BEGIN
   BB_G1.Bef.Bed_Res := FALSE;
   BB_G1.Bef.Bed_UV := FALSE;
   BB_G1.Bef.Bed_NHV := FALSE;
   BB_G1.Bef.Bed_PLS := FALSE;
   BB_G1.Bef.BA_Hand := FALSE;
   BB_G1.Bef.BA_Auto := FALSE;
   BB_G1.Bef.BF_Ein1 := FALSE;
   BB_G1.Bef.BF_Ein2 := FALSE;
   BB_G1.Bef.BF_Aus := FALSE;
   BB_G1.Bef.BZ_Res := FALSE;
   BB_G1.Bef.Res_10 := FALSE;
   BB_G1.Bef.Res_11 := FALSE;
   BB_G1.Bef.Res_12 := FALSE;
   BB_G1.Bef.Res_13 := FALSE;
   BB_G1.Bef.Res_14 := FALSE;
   BB_G1.Bef.Res_15 := FALSE;
   BB_G1.Bef.Res_16 := FALSE;
   BB_G1.Bef.Res_17 := FALSE;
   BB_G1.Bef.Res_18 := FALSE;
   BB_G1.Bef.Res_19 := FALSE;
   BB_G1.Bef.Res_20 := FALSE;
   BB_G1.Bef.Res_21 := FALSE;
   BB_G1.Bef.Res_22 := FALSE;
   BB_G1.Bef.Res_23 := FALSE;
   BB_G1.Bef.Res_24 := FALSE;
   BB_G1.Bef.Res_25 := FALSE;
   BB_G1.Bef.Res_26 := FALSE;
   BB_G1.Bef.Res_27 := FALSE;
   BB_G1.Bef.Res_28 := FALSE;
   BB_G1.Bef.Res_29 := FALSE;
   BB_G1.Bef.BF_Set_SW_chg := FALSE;
   BB_G1.Bef.BF_Quit := FALSE;
   BB_G1.SW_Hand := 0.0;
   BB_G2.Bef.Bed_Res := FALSE;
   BB_G2.Bef.Bed_UV := FALSE;
   BB_G2.Bef.Bed_NHV := FALSE;
   BB_G2.Bef.Bed_PLS := FALSE;
   BB_G2.Bef.BA_Hand := FALSE;
   BB_G2.Bef.BA_Auto := FALSE;
   BB_G2.Bef.BF_Ein1 := FALSE;
   BB_G2.Bef.BF_Ein2 := FALSE;
   BB_G2.Bef.BF_Aus := FALSE;
   BB_G2.Bef.BZ_Res := FALSE;
   BB_G2.Bef.Res_10 := FALSE;
   BB_G2.Bef.Res_11 := FALSE;
   BB_G2.Bef.Res_12 := FALSE;
   BB_G2.Bef.Res_13 := FALSE;
   BB_G2.Bef.Res_14 := FALSE;
   BB_G2.Bef.Res_15 := FALSE;
   BB_G2.Bef.Res_16 := FALSE;
   BB_G2.Bef.Res_17 := FALSE;
   BB_G2.Bef.Res_18 := FALSE;
   BB_G2.Bef.Res_19 := FALSE;
   BB_G2.Bef.Res_20 := FALSE;
   BB_G2.Bef.Res_21 := FALSE;
   BB_G2.Bef.Res_22 := FALSE;
   BB_G2.Bef.Res_23 := FALSE;
   BB_G2.Bef.Res_24 := FALSE;
   BB_G2.Bef.Res_25 := FALSE;
   BB_G2.Bef.Res_26 := FALSE;
   BB_G2.Bef.Res_27 := FALSE;
   BB_G2.Bef.Res_28 := FALSE;
   BB_G2.Bef.Res_29 := FALSE;
   BB_G2.Bef.BF_Set_SW_chg := FALSE;
   BB_G2.Bef.BF_Quit := FALSE;
   BB_G2.SW_Hand := 0.0;
   BB_G3.Bef.Bed_Res := FALSE;
   BB_G3.Bef.Bed_UV := FALSE;
   BB_G3.Bef.Bed_NHV := FALSE;
   BB_G3.Bef.Bed_PLS := FALSE;
   BB_G3.Bef.BA_Hand := FALSE;
   BB_G3.Bef.BA_Auto := FALSE;
   BB_G3.Bef.BF_Ein1 := FALSE;
   BB_G3.Bef.BF_Ein2 := FALSE;
   BB_G3.Bef.BF_Aus := FALSE;
   BB_G3.Bef.BZ_Res := FALSE;
   BB_G3.Bef.Res_10 := FALSE;
   BB_G3.Bef.Res_11 := FALSE;
   BB_G3.Bef.Res_12 := FALSE;
   BB_G3.Bef.Res_13 := FALSE;
   BB_G3.Bef.Res_14 := FALSE;
   BB_G3.Bef.Res_15 := FALSE;
   BB_G3.Bef.Res_16 := FALSE;
   BB_G3.Bef.Res_17 := FALSE;
   BB_G3.Bef.Res_18 := FALSE;
   BB_G3.Bef.Res_19 := FALSE;
   BB_G3.Bef.Res_20 := FALSE;
   BB_G3.Bef.Res_21 := FALSE;
   BB_G3.Bef.Res_22 := FALSE;
   BB_G3.Bef.Res_23 := FALSE;
   BB_G3.Bef.Res_24 := FALSE;
   BB_G3.Bef.Res_25 := FALSE;
   BB_G3.Bef.Res_26 := FALSE;
   BB_G3.Bef.Res_27 := FALSE;
   BB_G3.Bef.Res_28 := FALSE;
   BB_G3.Bef.Res_29 := FALSE;
   BB_G3.Bef.BF_Set_SW_chg := FALSE;
   BB_G3.Bef.BF_Quit := FALSE;
   BB_G3.SW_Hand := 0.0;
   BB_SHL_G1.Bef.Bed_Res := FALSE;
   BB_SHL_G1.Bef.Bed_UV := FALSE;
   BB_SHL_G1.Bef.Bed_NHV := FALSE;
   BB_SHL_G1.Bef.Bed_PLS := FALSE;
   BB_SHL_G1.Bef.BA_Hand := FALSE;
   BB_SHL_G1.Bef.BA_Auto := FALSE;
   BB_SHL_G1.Bef.BF_Ein1 := FALSE;
   BB_SHL_G1.Bef.BF_Ein2 := FALSE;
   BB_SHL_G1.Bef.BF_Aus := FALSE;
   BB_SHL_G1.Bef.BZ_Res := FALSE;
   BB_SHL_G1.Bef.Res_10 := FALSE;
   BB_SHL_G1.Bef.Res_11 := FALSE;
   BB_SHL_G1.Bef.Res_12 := FALSE;
   BB_SHL_G1.Bef.Res_13 := FALSE;
   BB_SHL_G1.Bef.Res_14 := FALSE;
   BB_SHL_G1.Bef.Res_15 := FALSE;
   BB_SHL_G1.Bef.Res_16 := FALSE;
   BB_SHL_G1.Bef.Res_17 := FALSE;
   BB_SHL_G1.Bef.Res_18 := FALSE;
   BB_SHL_G1.Bef.Res_19 := FALSE;
   BB_SHL_G1.Bef.Res_20 := FALSE;
   BB_SHL_G1.Bef.Res_21 := FALSE;
   BB_SHL_G1.Bef.Res_22 := FALSE;
   BB_SHL_G1.Bef.Res_23 := FALSE;
   BB_SHL_G1.Bef.Res_24 := FALSE;
   BB_SHL_G1.Bef.Res_25 := FALSE;
   BB_SHL_G1.Bef.Res_26 := FALSE;
   BB_SHL_G1.Bef.Res_27 := FALSE;
   BB_SHL_G1.Bef.Res_28 := FALSE;
   BB_SHL_G1.Bef.Res_29 := FALSE;
   BB_SHL_G1.Bef.BF_Set_SW_chg := FALSE;
   BB_SHL_G1.Bef.BF_Quit := FALSE;
   BB_SHL_G1.SW_Hand := 0.0;
   BB_SHL_G2.Bef.Bed_Res := FALSE;
   BB_SHL_G2.Bef.Bed_UV := FALSE;
   BB_SHL_G2.Bef.Bed_NHV := FALSE;
   BB_SHL_G2.Bef.Bed_PLS := FALSE;
   BB_SHL_G2.Bef.BA_Hand := FALSE;
   BB_SHL_G2.Bef.BA_Auto := FALSE;
   BB_SHL_G2.Bef.BF_Ein1 := FALSE;
   BB_SHL_G2.Bef.BF_Ein2 := FALSE;
   BB_SHL_G2.Bef.BF_Aus := FALSE;
   BB_SHL_G2.Bef.BZ_Res := FALSE;
   BB_SHL_G2.Bef.Res_10 := FALSE;
   BB_SHL_G2.Bef.Res_11 := FALSE;
   BB_SHL_G2.Bef.Res_12 := FALSE;
   BB_SHL_G2.Bef.Res_13 := FALSE;
   BB_SHL_G2.Bef.Res_14 := FALSE;
   BB_SHL_G2.Bef.Res_15 := FALSE;
   BB_SHL_G2.Bef.Res_16 := FALSE;
   BB_SHL_G2.Bef.Res_17 := FALSE;
   BB_SHL_G2.Bef.Res_18 := FALSE;
   BB_SHL_G2.Bef.Res_19 := FALSE;
   BB_SHL_G2.Bef.Res_20 := FALSE;
   BB_SHL_G2.Bef.Res_21 := FALSE;
   BB_SHL_G2.Bef.Res_22 := FALSE;
   BB_SHL_G2.Bef.Res_23 := FALSE;
   BB_SHL_G2.Bef.Res_24 := FALSE;
   BB_SHL_G2.Bef.Res_25 := FALSE;
   BB_SHL_G2.Bef.Res_26 := FALSE;
   BB_SHL_G2.Bef.Res_27 := FALSE;
   BB_SHL_G2.Bef.Res_28 := FALSE;
   BB_SHL_G2.Bef.Res_29 := FALSE;
   BB_SHL_G2.Bef.BF_Set_SW_chg := FALSE;
   BB_SHL_G2.Bef.BF_Quit := FALSE;
   BB_SHL_G2.SW_Hand := 0.0;
   BB_SHL_G3.Bef.Bed_Res := FALSE;
   BB_SHL_G3.Bef.Bed_UV := FALSE;
   BB_SHL_G3.Bef.Bed_NHV := FALSE;
   BB_SHL_G3.Bef.Bed_PLS := FALSE;
   BB_SHL_G3.Bef.BA_Hand := FALSE;
   BB_SHL_G3.Bef.BA_Auto := FALSE;
   BB_SHL_G3.Bef.BF_Ein1 := FALSE;
   BB_SHL_G3.Bef.BF_Ein2 := FALSE;
   BB_SHL_G3.Bef.BF_Aus := FALSE;
   BB_SHL_G3.Bef.BZ_Res := FALSE;
   BB_SHL_G3.Bef.Res_10 := FALSE;
   BB_SHL_G3.Bef.Res_11 := FALSE;
   BB_SHL_G3.Bef.Res_12 := FALSE;
   BB_SHL_G3.Bef.Res_13 := FALSE;
   BB_SHL_G3.Bef.Res_14 := FALSE;
   BB_SHL_G3.Bef.Res_15 := FALSE;
   BB_SHL_G3.Bef.Res_16 := FALSE;
   BB_SHL_G3.Bef.Res_17 := FALSE;
   BB_SHL_G3.Bef.Res_18 := FALSE;
   BB_SHL_G3.Bef.Res_19 := FALSE;
   BB_SHL_G3.Bef.Res_20 := FALSE;
   BB_SHL_G3.Bef.Res_21 := FALSE;
   BB_SHL_G3.Bef.Res_22 := FALSE;
   BB_SHL_G3.Bef.Res_23 := FALSE;
   BB_SHL_G3.Bef.Res_24 := FALSE;
   BB_SHL_G3.Bef.Res_25 := FALSE;
   BB_SHL_G3.Bef.Res_26 := FALSE;
   BB_SHL_G3.Bef.Res_27 := FALSE;
   BB_SHL_G3.Bef.Res_28 := FALSE;
   BB_SHL_G3.Bef.Res_29 := FALSE;
   BB_SHL_G3.Bef.BF_Set_SW_chg := FALSE;
   BB_SHL_G3.Bef.BF_Quit := FALSE;
   BB_SHL_G3.SW_Hand := 0.0;
   BB_AV.Bef.Bed_Res := FALSE;
   BB_AV.Bef.Bed_UV := FALSE;
   BB_AV.Bef.Bed_NHV := FALSE;
   BB_AV.Bef.Bed_PLS := FALSE;
   BB_AV.Bef.BA_Hand := FALSE;
   BB_AV.Bef.BA_Auto := FALSE;
   BB_AV.Bef.BF_Ein1 := FALSE;
   BB_AV.Bef.BF_Ein2 := FALSE;
   BB_AV.Bef.BF_Aus := FALSE;
   BB_AV.Bef.BZ_Res := FALSE;
   BB_AV.Bef.Res_10 := FALSE;
   BB_AV.Bef.Res_11 := FALSE;
   BB_AV.Bef.Res_12 := FALSE;
   BB_AV.Bef.Res_13 := FALSE;
   BB_AV.Bef.Res_14 := FALSE;
   BB_AV.Bef.Res_15 := FALSE;
   BB_AV.Bef.Res_16 := FALSE;
   BB_AV.Bef.Res_17 := FALSE;
   BB_AV.Bef.Res_18 := FALSE;
   BB_AV.Bef.Res_19 := FALSE;
   BB_AV.Bef.Res_20 := FALSE;
   BB_AV.Bef.Res_21 := FALSE;
   BB_AV.Bef.Res_22 := FALSE;
   BB_AV.Bef.Res_23 := FALSE;
   BB_AV.Bef.Res_24 := FALSE;
   BB_AV.Bef.Res_25 := FALSE;
   BB_AV.Bef.Res_26 := FALSE;
   BB_AV.Bef.Res_27 := FALSE;
   BB_AV.Bef.Res_28 := FALSE;
   BB_AV.Bef.Res_29 := FALSE;
   BB_AV.Bef.BF_Set_SW_chg := FALSE;
   BB_AV.Bef.BF_Quit := FALSE;
   BB_AV.SW_Hand := 0.0;
   BB_LS1.Bef.Bed_Res := FALSE;
   BB_LS1.Bef.Bed_UV := FALSE;
   BB_LS1.Bef.Bed_NHV := FALSE;
   BB_LS1.Bef.Bed_PLS := FALSE;
   BB_LS1.Bef.BA_Hand := FALSE;
   BB_LS1.Bef.BA_Auto := FALSE;
   BB_LS1.Bef.BF_Ein1 := FALSE;
   BB_LS1.Bef.BF_Ein2 := FALSE;
   BB_LS1.Bef.BF_Aus := FALSE;
   BB_LS1.Bef.BZ_Res := FALSE;
   BB_LS1.Bef.Res_10 := FALSE;
   BB_LS1.Bef.Res_11 := FALSE;
   BB_LS1.Bef.Res_12 := FALSE;
   BB_LS1.Bef.Res_13 := FALSE;
   BB_LS1.Bef.Res_14 := FALSE;
   BB_LS1.Bef.Res_15 := FALSE;
   BB_LS1.Bef.Res_16 := FALSE;
   BB_LS1.Bef.Res_17 := FALSE;
   BB_LS1.Bef.Res_18 := FALSE;
   BB_LS1.Bef.Res_19 := FALSE;
   BB_LS1.Bef.Res_20 := FALSE;
   BB_LS1.Bef.Res_21 := FALSE;
   BB_LS1.Bef.Res_22 := FALSE;
   BB_LS1.Bef.Res_23 := FALSE;
   BB_LS1.Bef.Res_24 := FALSE;
   BB_LS1.Bef.Res_25 := FALSE;
   BB_LS1.Bef.Res_26 := FALSE;
   BB_LS1.Bef.Res_27 := FALSE;
   BB_LS1.Bef.Res_28 := FALSE;
   BB_LS1.Bef.Res_29 := FALSE;
   BB_LS1.Bef.BF_Set_SW_chg := FALSE;
   BB_LS1.Bef.BF_Quit := FALSE;
   BB_LS1.SW_Hand := 0.0;
   BB_LS2.Bef.Bed_Res := FALSE;
   BB_LS2.Bef.Bed_UV := FALSE;
   BB_LS2.Bef.Bed_NHV := FALSE;
   BB_LS2.Bef.Bed_PLS := FALSE;
   BB_LS2.Bef.BA_Hand := FALSE;
   BB_LS2.Bef.BA_Auto := FALSE;
   BB_LS2.Bef.BF_Ein1 := FALSE;
   BB_LS2.Bef.BF_Ein2 := FALSE;
   BB_LS2.Bef.BF_Aus := FALSE;
   BB_LS2.Bef.BZ_Res := FALSE;
   BB_LS2.Bef.Res_10 := FALSE;
   BB_LS2.Bef.Res_11 := FALSE;
   BB_LS2.Bef.Res_12 := FALSE;
   BB_LS2.Bef.Res_13 := FALSE;
   BB_LS2.Bef.Res_14 := FALSE;
   BB_LS2.Bef.Res_15 := FALSE;
   BB_LS2.Bef.Res_16 := FALSE;
   BB_LS2.Bef.Res_17 := FALSE;
   BB_LS2.Bef.Res_18 := FALSE;
   BB_LS2.Bef.Res_19 := FALSE;
   BB_LS2.Bef.Res_20 := FALSE;
   BB_LS2.Bef.Res_21 := FALSE;
   BB_LS2.Bef.Res_22 := FALSE;
   BB_LS2.Bef.Res_23 := FALSE;
   BB_LS2.Bef.Res_24 := FALSE;
   BB_LS2.Bef.Res_25 := FALSE;
   BB_LS2.Bef.Res_26 := FALSE;
   BB_LS2.Bef.Res_27 := FALSE;
   BB_LS2.Bef.Res_28 := FALSE;
   BB_LS2.Bef.Res_29 := FALSE;
   BB_LS2.Bef.BF_Set_SW_chg := FALSE;
   BB_LS2.Bef.BF_Quit := FALSE;
   BB_LS2.SW_Hand := 0.0;
   BB1_RZP1.Bef.Bed_Res := FALSE;
   BB1_RZP1.Bef.Bed_UV := FALSE;
   BB1_RZP1.Bef.Bed_NHV := FALSE;
   BB1_RZP1.Bef.Bed_PLS := FALSE;
   BB1_RZP1.Bef.BA_Hand := FALSE;
   BB1_RZP1.Bef.BA_Auto := FALSE;
   BB1_RZP1.Bef.BF_Ein1 := FALSE;
   BB1_RZP1.Bef.BF_Ein2 := FALSE;
   BB1_RZP1.Bef.BF_Aus := FALSE;
   BB1_RZP1.Bef.BZ_Res := FALSE;
   BB1_RZP1.Bef.Res_10 := FALSE;
   BB1_RZP1.Bef.Res_11 := FALSE;
   BB1_RZP1.Bef.Res_12 := FALSE;
   BB1_RZP1.Bef.Res_13 := FALSE;
   BB1_RZP1.Bef.Res_14 := FALSE;
   BB1_RZP1.Bef.Res_15 := FALSE;
   BB1_RZP1.Bef.Res_16 := FALSE;
   BB1_RZP1.Bef.Res_17 := FALSE;
   BB1_RZP1.Bef.Res_18 := FALSE;
   BB1_RZP1.Bef.Res_19 := FALSE;
   BB1_RZP1.Bef.Res_20 := FALSE;
   BB1_RZP1.Bef.Res_21 := FALSE;
   BB1_RZP1.Bef.Res_22 := FALSE;
   BB1_RZP1.Bef.Res_23 := FALSE;
   BB1_RZP1.Bef.Res_24 := FALSE;
   BB1_RZP1.Bef.Res_25 := FALSE;
   BB1_RZP1.Bef.Res_26 := FALSE;
   BB1_RZP1.Bef.Res_27 := FALSE;
   BB1_RZP1.Bef.Res_28 := FALSE;
   BB1_RZP1.Bef.Res_29 := FALSE;
   BB1_RZP1.Bef.BF_Set_SW_chg := FALSE;
   BB1_RZP1.Bef.BF_Quit := FALSE;
   BB1_RZP1.SW_Hand := 0.0;
   BB1_RZP2.Bef.Bed_Res := FALSE;
   BB1_RZP2.Bef.Bed_UV := FALSE;
   BB1_RZP2.Bef.Bed_NHV := FALSE;
   BB1_RZP2.Bef.Bed_PLS := FALSE;
   BB1_RZP2.Bef.BA_Hand := FALSE;
   BB1_RZP2.Bef.BA_Auto := FALSE;
   BB1_RZP2.Bef.BF_Ein1 := FALSE;
   BB1_RZP2.Bef.BF_Ein2 := FALSE;
   BB1_RZP2.Bef.BF_Aus := FALSE;
   BB1_RZP2.Bef.BZ_Res := FALSE;
   BB1_RZP2.Bef.Res_10 := FALSE;
   BB1_RZP2.Bef.Res_11 := FALSE;
   BB1_RZP2.Bef.Res_12 := FALSE;
   BB1_RZP2.Bef.Res_13 := FALSE;
   BB1_RZP2.Bef.Res_14 := FALSE;
   BB1_RZP2.Bef.Res_15 := FALSE;
   BB1_RZP2.Bef.Res_16 := FALSE;
   BB1_RZP2.Bef.Res_17 := FALSE;
   BB1_RZP2.Bef.Res_18 := FALSE;
   BB1_RZP2.Bef.Res_19 := FALSE;
   BB1_RZP2.Bef.Res_20 := FALSE;
   BB1_RZP2.Bef.Res_21 := FALSE;
   BB1_RZP2.Bef.Res_22 := FALSE;
   BB1_RZP2.Bef.Res_23 := FALSE;
   BB1_RZP2.Bef.Res_24 := FALSE;
   BB1_RZP2.Bef.Res_25 := FALSE;
   BB1_RZP2.Bef.Res_26 := FALSE;
   BB1_RZP2.Bef.Res_27 := FALSE;
   BB1_RZP2.Bef.Res_28 := FALSE;
   BB1_RZP2.Bef.Res_29 := FALSE;
   BB1_RZP2.Bef.BF_Set_SW_chg := FALSE;
   BB1_RZP2.Bef.BF_Quit := FALSE;
   BB1_RZP2.SW_Hand := 0.0;
   BB1_UeSP.Bef.Bed_Res := FALSE;
   BB1_UeSP.Bef.Bed_UV := FALSE;
   BB1_UeSP.Bef.Bed_NHV := FALSE;
   BB1_UeSP.Bef.Bed_PLS := FALSE;
   BB1_UeSP.Bef.BA_Hand := FALSE;
   BB1_UeSP.Bef.BA_Auto := FALSE;
   BB1_UeSP.Bef.BF_Ein1 := FALSE;
   BB1_UeSP.Bef.BF_Ein2 := FALSE;
   BB1_UeSP.Bef.BF_Aus := FALSE;
   BB1_UeSP.Bef.BZ_Res := FALSE;
   BB1_UeSP.Bef.Res_10 := FALSE;
   BB1_UeSP.Bef.Res_11 := FALSE;
   BB1_UeSP.Bef.Res_12 := FALSE;
   BB1_UeSP.Bef.Res_13 := FALSE;
   BB1_UeSP.Bef.Res_14 := FALSE;
   BB1_UeSP.Bef.Res_15 := FALSE;
   BB1_UeSP.Bef.Res_16 := FALSE;
   BB1_UeSP.Bef.Res_17 := FALSE;
   BB1_UeSP.Bef.Res_18 := FALSE;
   BB1_UeSP.Bef.Res_19 := FALSE;
   BB1_UeSP.Bef.Res_20 := FALSE;
   BB1_UeSP.Bef.Res_21 := FALSE;
   BB1_UeSP.Bef.Res_22 := FALSE;
   BB1_UeSP.Bef.Res_23 := FALSE;
   BB1_UeSP.Bef.Res_24 := FALSE;
   BB1_UeSP.Bef.Res_25 := FALSE;
   BB1_UeSP.Bef.Res_26 := FALSE;
   BB1_UeSP.Bef.Res_27 := FALSE;
   BB1_UeSP.Bef.Res_28 := FALSE;
   BB1_UeSP.Bef.Res_29 := FALSE;
   BB1_UeSP.Bef.BF_Set_SW_chg := FALSE;
   BB1_UeSP.Bef.BF_Quit := FALSE;
   BB1_UeSP.SW_Hand := 0.0;
   BB1_AS1.Bef.Bed_Res := FALSE;
   BB1_AS1.Bef.Bed_UV := FALSE;
   BB1_AS1.Bef.Bed_NHV := FALSE;
   BB1_AS1.Bef.Bed_PLS := FALSE;
   BB1_AS1.Bef.BA_Hand := FALSE;
   BB1_AS1.Bef.BA_Auto := FALSE;
   BB1_AS1.Bef.BF_Ein1 := FALSE;
   BB1_AS1.Bef.BF_Ein2 := FALSE;
   BB1_AS1.Bef.BF_Aus := FALSE;
   BB1_AS1.Bef.BZ_Res := FALSE;
   BB1_AS1.Bef.Res_10 := FALSE;
   BB1_AS1.Bef.Res_11 := FALSE;
   BB1_AS1.Bef.Res_12 := FALSE;
   BB1_AS1.Bef.Res_13 := FALSE;
   BB1_AS1.Bef.Res_14 := FALSE;
   BB1_AS1.Bef.Res_15 := FALSE;
   BB1_AS1.Bef.Res_16 := FALSE;
   BB1_AS1.Bef.Res_17 := FALSE;
   BB1_AS1.Bef.Res_18 := FALSE;
   BB1_AS1.Bef.Res_19 := FALSE;
   BB1_AS1.Bef.Res_20 := FALSE;
   BB1_AS1.Bef.Res_21 := FALSE;
   BB1_AS1.Bef.Res_22 := FALSE;
   BB1_AS1.Bef.Res_23 := FALSE;
   BB1_AS1.Bef.Res_24 := FALSE;
   BB1_AS1.Bef.Res_25 := FALSE;
   BB1_AS1.Bef.Res_26 := FALSE;
   BB1_AS1.Bef.Res_27 := FALSE;
   BB1_AS1.Bef.Res_28 := FALSE;
   BB1_AS1.Bef.Res_29 := FALSE;
   BB1_AS1.Bef.BF_Set_SW_chg := FALSE;
   BB1_AS1.Bef.BF_Quit := FALSE;
   BB1_AS1.SW_Hand := 0.0;
   BB1_AS2.Bef.Bed_Res := FALSE;
   BB1_AS2.Bef.Bed_UV := FALSE;
   BB1_AS2.Bef.Bed_NHV := FALSE;
   BB1_AS2.Bef.Bed_PLS := FALSE;
   BB1_AS2.Bef.BA_Hand := FALSE;
   BB1_AS2.Bef.BA_Auto := FALSE;
   BB1_AS2.Bef.BF_Ein1 := FALSE;
   BB1_AS2.Bef.BF_Ein2 := FALSE;
   BB1_AS2.Bef.BF_Aus := FALSE;
   BB1_AS2.Bef.BZ_Res := FALSE;
   BB1_AS2.Bef.Res_10 := FALSE;
   BB1_AS2.Bef.Res_11 := FALSE;
   BB1_AS2.Bef.Res_12 := FALSE;
   BB1_AS2.Bef.Res_13 := FALSE;
   BB1_AS2.Bef.Res_14 := FALSE;
   BB1_AS2.Bef.Res_15 := FALSE;
   BB1_AS2.Bef.Res_16 := FALSE;
   BB1_AS2.Bef.Res_17 := FALSE;
   BB1_AS2.Bef.Res_18 := FALSE;
   BB1_AS2.Bef.Res_19 := FALSE;
   BB1_AS2.Bef.Res_20 := FALSE;
   BB1_AS2.Bef.Res_21 := FALSE;
   BB1_AS2.Bef.Res_22 := FALSE;
   BB1_AS2.Bef.Res_23 := FALSE;
   BB1_AS2.Bef.Res_24 := FALSE;
   BB1_AS2.Bef.Res_25 := FALSE;
   BB1_AS2.Bef.Res_26 := FALSE;
   BB1_AS2.Bef.Res_27 := FALSE;
   BB1_AS2.Bef.Res_28 := FALSE;
   BB1_AS2.Bef.Res_29 := FALSE;
   BB1_AS2.Bef.BF_Set_SW_chg := FALSE;
   BB1_AS2.Bef.BF_Quit := FALSE;
   BB1_AS2.SW_Hand := 0.0;
   BB1_SR1.Bef.Bed_Res := FALSE;
   BB1_SR1.Bef.Bed_UV := FALSE;
   BB1_SR1.Bef.Bed_NHV := FALSE;
   BB1_SR1.Bef.Bed_PLS := FALSE;
   BB1_SR1.Bef.BA_Hand := FALSE;
   BB1_SR1.Bef.BA_Auto := FALSE;
   BB1_SR1.Bef.BF_Ein1 := FALSE;
   BB1_SR1.Bef.BF_Ein2 := FALSE;
   BB1_SR1.Bef.BF_Aus := FALSE;
   BB1_SR1.Bef.BZ_Res := FALSE;
   BB1_SR1.Bef.Res_10 := FALSE;
   BB1_SR1.Bef.Res_11 := FALSE;
   BB1_SR1.Bef.Res_12 := FALSE;
   BB1_SR1.Bef.Res_13 := FALSE;
   BB1_SR1.Bef.Res_14 := FALSE;
   BB1_SR1.Bef.Res_15 := FALSE;
   BB1_SR1.Bef.Res_16 := FALSE;
   BB1_SR1.Bef.Res_17 := FALSE;
   BB1_SR1.Bef.Res_18 := FALSE;
   BB1_SR1.Bef.Res_19 := FALSE;
   BB1_SR1.Bef.Res_20 := FALSE;
   BB1_SR1.Bef.Res_21 := FALSE;
   BB1_SR1.Bef.Res_22 := FALSE;
   BB1_SR1.Bef.Res_23 := FALSE;
   BB1_SR1.Bef.Res_24 := FALSE;
   BB1_SR1.Bef.Res_25 := FALSE;
   BB1_SR1.Bef.Res_26 := FALSE;
   BB1_SR1.Bef.Res_27 := FALSE;
   BB1_SR1.Bef.Res_28 := FALSE;
   BB1_SR1.Bef.Res_29 := FALSE;
   BB1_SR1.Bef.BF_Set_SW_chg := FALSE;
   BB1_SR1.Bef.BF_Quit := FALSE;
   BB1_SR1.SW_Hand := 0.0;
   BB1_SR2.Bef.Bed_Res := FALSE;
   BB1_SR2.Bef.Bed_UV := FALSE;
   BB1_SR2.Bef.Bed_NHV := FALSE;
   BB1_SR2.Bef.Bed_PLS := FALSE;
   BB1_SR2.Bef.BA_Hand := FALSE;
   BB1_SR2.Bef.BA_Auto := FALSE;
   BB1_SR2.Bef.BF_Ein1 := FALSE;
   BB1_SR2.Bef.BF_Ein2 := FALSE;
   BB1_SR2.Bef.BF_Aus := FALSE;
   BB1_SR2.Bef.BZ_Res := FALSE;
   BB1_SR2.Bef.Res_10 := FALSE;
   BB1_SR2.Bef.Res_11 := FALSE;
   BB1_SR2.Bef.Res_12 := FALSE;
   BB1_SR2.Bef.Res_13 := FALSE;
   BB1_SR2.Bef.Res_14 := FALSE;
   BB1_SR2.Bef.Res_15 := FALSE;
   BB1_SR2.Bef.Res_16 := FALSE;
   BB1_SR2.Bef.Res_17 := FALSE;
   BB1_SR2.Bef.Res_18 := FALSE;
   BB1_SR2.Bef.Res_19 := FALSE;
   BB1_SR2.Bef.Res_20 := FALSE;
   BB1_SR2.Bef.Res_21 := FALSE;
   BB1_SR2.Bef.Res_22 := FALSE;
   BB1_SR2.Bef.Res_23 := FALSE;
   BB1_SR2.Bef.Res_24 := FALSE;
   BB1_SR2.Bef.Res_25 := FALSE;
   BB1_SR2.Bef.Res_26 := FALSE;
   BB1_SR2.Bef.Res_27 := FALSE;
   BB1_SR2.Bef.Res_28 := FALSE;
   BB1_SR2.Bef.Res_29 := FALSE;
   BB1_SR2.Bef.BF_Set_SW_chg := FALSE;
   BB1_SR2.Bef.BF_Quit := FALSE;
   BB1_SR2.SW_Hand := 0.0;
   BB2_RZP1.Bef.Bed_Res := FALSE;
   BB2_RZP1.Bef.Bed_UV := FALSE;
   BB2_RZP1.Bef.Bed_NHV := FALSE;
   BB2_RZP1.Bef.Bed_PLS := FALSE;
   BB2_RZP1.Bef.BA_Hand := FALSE;
   BB2_RZP1.Bef.BA_Auto := FALSE;
   BB2_RZP1.Bef.BF_Ein1 := FALSE;
   BB2_RZP1.Bef.BF_Ein2 := FALSE;
   BB2_RZP1.Bef.BF_Aus := FALSE;
   BB2_RZP1.Bef.BZ_Res := FALSE;
   BB2_RZP1.Bef.Res_10 := FALSE;
   BB2_RZP1.Bef.Res_11 := FALSE;
   BB2_RZP1.Bef.Res_12 := FALSE;
   BB2_RZP1.Bef.Res_13 := FALSE;
   BB2_RZP1.Bef.Res_14 := FALSE;
   BB2_RZP1.Bef.Res_15 := FALSE;
   BB2_RZP1.Bef.Res_16 := FALSE;
   BB2_RZP1.Bef.Res_17 := FALSE;
   BB2_RZP1.Bef.Res_18 := FALSE;
   BB2_RZP1.Bef.Res_19 := FALSE;
   BB2_RZP1.Bef.Res_20 := FALSE;
   BB2_RZP1.Bef.Res_21 := FALSE;
   BB2_RZP1.Bef.Res_22 := FALSE;
   BB2_RZP1.Bef.Res_23 := FALSE;
   BB2_RZP1.Bef.Res_24 := FALSE;
   BB2_RZP1.Bef.Res_25 := FALSE;
   BB2_RZP1.Bef.Res_26 := FALSE;
   BB2_RZP1.Bef.Res_27 := FALSE;
   BB2_RZP1.Bef.Res_28 := FALSE;
   BB2_RZP1.Bef.Res_29 := FALSE;
   BB2_RZP1.Bef.BF_Set_SW_chg := FALSE;
   BB2_RZP1.Bef.BF_Quit := FALSE;
   BB2_RZP1.SW_Hand := 0.0;
   BB2_RZP2.Bef.Bed_Res := FALSE;
   BB2_RZP2.Bef.Bed_UV := FALSE;
   BB2_RZP2.Bef.Bed_NHV := FALSE;
   BB2_RZP2.Bef.Bed_PLS := FALSE;
   BB2_RZP2.Bef.BA_Hand := FALSE;
   BB2_RZP2.Bef.BA_Auto := FALSE;
   BB2_RZP2.Bef.BF_Ein1 := FALSE;
   BB2_RZP2.Bef.BF_Ein2 := FALSE;
   BB2_RZP2.Bef.BF_Aus := FALSE;
   BB2_RZP2.Bef.BZ_Res := FALSE;
   BB2_RZP2.Bef.Res_10 := FALSE;
   BB2_RZP2.Bef.Res_11 := FALSE;
   BB2_RZP2.Bef.Res_12 := FALSE;
   BB2_RZP2.Bef.Res_13 := FALSE;
   BB2_RZP2.Bef.Res_14 := FALSE;
   BB2_RZP2.Bef.Res_15 := FALSE;
   BB2_RZP2.Bef.Res_16 := FALSE;
   BB2_RZP2.Bef.Res_17 := FALSE;
   BB2_RZP2.Bef.Res_18 := FALSE;
   BB2_RZP2.Bef.Res_19 := FALSE;
   BB2_RZP2.Bef.Res_20 := FALSE;
   BB2_RZP2.Bef.Res_21 := FALSE;
   BB2_RZP2.Bef.Res_22 := FALSE;
   BB2_RZP2.Bef.Res_23 := FALSE;
   BB2_RZP2.Bef.Res_24 := FALSE;
   BB2_RZP2.Bef.Res_25 := FALSE;
   BB2_RZP2.Bef.Res_26 := FALSE;
   BB2_RZP2.Bef.Res_27 := FALSE;
   BB2_RZP2.Bef.Res_28 := FALSE;
   BB2_RZP2.Bef.Res_29 := FALSE;
   BB2_RZP2.Bef.BF_Set_SW_chg := FALSE;
   BB2_RZP2.Bef.BF_Quit := FALSE;
   BB2_RZP2.SW_Hand := 0.0;
   BB2_UeSP.Bef.Bed_Res := FALSE;
   BB2_UeSP.Bef.Bed_UV := FALSE;
   BB2_UeSP.Bef.Bed_NHV := FALSE;
   BB2_UeSP.Bef.Bed_PLS := FALSE;
   BB2_UeSP.Bef.BA_Hand := FALSE;
   BB2_UeSP.Bef.BA_Auto := FALSE;
   BB2_UeSP.Bef.BF_Ein1 := FALSE;
   BB2_UeSP.Bef.BF_Ein2 := FALSE;
   BB2_UeSP.Bef.BF_Aus := FALSE;
   BB2_UeSP.Bef.BZ_Res := FALSE;
   BB2_UeSP.Bef.Res_10 := FALSE;
   BB2_UeSP.Bef.Res_11 := FALSE;
   BB2_UeSP.Bef.Res_12 := FALSE;
   BB2_UeSP.Bef.Res_13 := FALSE;
   BB2_UeSP.Bef.Res_14 := FALSE;
   BB2_UeSP.Bef.Res_15 := FALSE;
   BB2_UeSP.Bef.Res_16 := FALSE;
   BB2_UeSP.Bef.Res_17 := FALSE;
   BB2_UeSP.Bef.Res_18 := FALSE;
   BB2_UeSP.Bef.Res_19 := FALSE;
   BB2_UeSP.Bef.Res_20 := FALSE;
   BB2_UeSP.Bef.Res_21 := FALSE;
   BB2_UeSP.Bef.Res_22 := FALSE;
   BB2_UeSP.Bef.Res_23 := FALSE;
   BB2_UeSP.Bef.Res_24 := FALSE;
   BB2_UeSP.Bef.Res_25 := FALSE;
   BB2_UeSP.Bef.Res_26 := FALSE;
   BB2_UeSP.Bef.Res_27 := FALSE;
   BB2_UeSP.Bef.Res_28 := FALSE;
   BB2_UeSP.Bef.Res_29 := FALSE;
   BB2_UeSP.Bef.BF_Set_SW_chg := FALSE;
   BB2_UeSP.Bef.BF_Quit := FALSE;
   BB2_UeSP.SW_Hand := 0.0;
   BB2_AS1.Bef.Bed_Res := FALSE;
   BB2_AS1.Bef.Bed_UV := FALSE;
   BB2_AS1.Bef.Bed_NHV := FALSE;
   BB2_AS1.Bef.Bed_PLS := FALSE;
   BB2_AS1.Bef.BA_Hand := FALSE;
   BB2_AS1.Bef.BA_Auto := FALSE;
   BB2_AS1.Bef.BF_Ein1 := FALSE;
   BB2_AS1.Bef.BF_Ein2 := FALSE;
   BB2_AS1.Bef.BF_Aus := FALSE;
   BB2_AS1.Bef.BZ_Res := FALSE;
   BB2_AS1.Bef.Res_10 := FALSE;
   BB2_AS1.Bef.Res_11 := FALSE;
   BB2_AS1.Bef.Res_12 := FALSE;
   BB2_AS1.Bef.Res_13 := FALSE;
   BB2_AS1.Bef.Res_14 := FALSE;
   BB2_AS1.Bef.Res_15 := FALSE;
   BB2_AS1.Bef.Res_16 := FALSE;
   BB2_AS1.Bef.Res_17 := FALSE;
   BB2_AS1.Bef.Res_18 := FALSE;
   BB2_AS1.Bef.Res_19 := FALSE;
   BB2_AS1.Bef.Res_20 := FALSE;
   BB2_AS1.Bef.Res_21 := FALSE;
   BB2_AS1.Bef.Res_22 := FALSE;
   BB2_AS1.Bef.Res_23 := FALSE;
   BB2_AS1.Bef.Res_24 := FALSE;
   BB2_AS1.Bef.Res_25 := FALSE;
   BB2_AS1.Bef.Res_26 := FALSE;
   BB2_AS1.Bef.Res_27 := FALSE;
   BB2_AS1.Bef.Res_28 := FALSE;
   BB2_AS1.Bef.Res_29 := FALSE;
   BB2_AS1.Bef.BF_Set_SW_chg := FALSE;
   BB2_AS1.Bef.BF_Quit := FALSE;
   BB2_AS1.SW_Hand := 0.0;
   BB2_AS2.Bef.Bed_Res := FALSE;
   BB2_AS2.Bef.Bed_UV := FALSE;
   BB2_AS2.Bef.Bed_NHV := FALSE;
   BB2_AS2.Bef.Bed_PLS := FALSE;
   BB2_AS2.Bef.BA_Hand := FALSE;
   BB2_AS2.Bef.BA_Auto := FALSE;
   BB2_AS2.Bef.BF_Ein1 := FALSE;
   BB2_AS2.Bef.BF_Ein2 := FALSE;
   BB2_AS2.Bef.BF_Aus := FALSE;
   BB2_AS2.Bef.BZ_Res := FALSE;
   BB2_AS2.Bef.Res_10 := FALSE;
   BB2_AS2.Bef.Res_11 := FALSE;
   BB2_AS2.Bef.Res_12 := FALSE;
   BB2_AS2.Bef.Res_13 := FALSE;
   BB2_AS2.Bef.Res_14 := FALSE;
   BB2_AS2.Bef.Res_15 := FALSE;
   BB2_AS2.Bef.Res_16 := FALSE;
   BB2_AS2.Bef.Res_17 := FALSE;
   BB2_AS2.Bef.Res_18 := FALSE;
   BB2_AS2.Bef.Res_19 := FALSE;
   BB2_AS2.Bef.Res_20 := FALSE;
   BB2_AS2.Bef.Res_21 := FALSE;
   BB2_AS2.Bef.Res_22 := FALSE;
   BB2_AS2.Bef.Res_23 := FALSE;
   BB2_AS2.Bef.Res_24 := FALSE;
   BB2_AS2.Bef.Res_25 := FALSE;
   BB2_AS2.Bef.Res_26 := FALSE;
   BB2_AS2.Bef.Res_27 := FALSE;
   BB2_AS2.Bef.Res_28 := FALSE;
   BB2_AS2.Bef.Res_29 := FALSE;
   BB2_AS2.Bef.BF_Set_SW_chg := FALSE;
   BB2_AS2.Bef.BF_Quit := FALSE;
   BB2_AS2.SW_Hand := 0.0;
   BB2_SR1.Bef.Bed_Res := FALSE;
   BB2_SR1.Bef.Bed_UV := FALSE;
   BB2_SR1.Bef.Bed_NHV := FALSE;
   BB2_SR1.Bef.Bed_PLS := FALSE;
   BB2_SR1.Bef.BA_Hand := FALSE;
   BB2_SR1.Bef.BA_Auto := FALSE;
   BB2_SR1.Bef.BF_Ein1 := FALSE;
   BB2_SR1.Bef.BF_Ein2 := FALSE;
   BB2_SR1.Bef.BF_Aus := FALSE;
   BB2_SR1.Bef.BZ_Res := FALSE;
   BB2_SR1.Bef.Res_10 := FALSE;
   BB2_SR1.Bef.Res_11 := FALSE;
   BB2_SR1.Bef.Res_12 := FALSE;
   BB2_SR1.Bef.Res_13 := FALSE;
   BB2_SR1.Bef.Res_14 := FALSE;
   BB2_SR1.Bef.Res_15 := FALSE;
   BB2_SR1.Bef.Res_16 := FALSE;
   BB2_SR1.Bef.Res_17 := FALSE;
   BB2_SR1.Bef.Res_18 := FALSE;
   BB2_SR1.Bef.Res_19 := FALSE;
   BB2_SR1.Bef.Res_20 := FALSE;
   BB2_SR1.Bef.Res_21 := FALSE;
   BB2_SR1.Bef.Res_22 := FALSE;
   BB2_SR1.Bef.Res_23 := FALSE;
   BB2_SR1.Bef.Res_24 := FALSE;
   BB2_SR1.Bef.Res_25 := FALSE;
   BB2_SR1.Bef.Res_26 := FALSE;
   BB2_SR1.Bef.Res_27 := FALSE;
   BB2_SR1.Bef.Res_28 := FALSE;
   BB2_SR1.Bef.Res_29 := FALSE;
   BB2_SR1.Bef.BF_Set_SW_chg := TRUE;
   BB2_SR1.Bef.BF_Quit := FALSE;
   BB2_SR1.SW_Hand := 0.0;
   BB2_SR2.Bef.Bed_Res := FALSE;
   BB2_SR2.Bef.Bed_UV := FALSE;
   BB2_SR2.Bef.Bed_NHV := FALSE;
   BB2_SR2.Bef.Bed_PLS := FALSE;
   BB2_SR2.Bef.BA_Hand := FALSE;
   BB2_SR2.Bef.BA_Auto := FALSE;
   BB2_SR2.Bef.BF_Ein1 := FALSE;
   BB2_SR2.Bef.BF_Ein2 := FALSE;
   BB2_SR2.Bef.BF_Aus := FALSE;
   BB2_SR2.Bef.BZ_Res := FALSE;
   BB2_SR2.Bef.Res_10 := FALSE;
   BB2_SR2.Bef.Res_11 := FALSE;
   BB2_SR2.Bef.Res_12 := FALSE;
   BB2_SR2.Bef.Res_13 := FALSE;
   BB2_SR2.Bef.Res_14 := FALSE;
   BB2_SR2.Bef.Res_15 := FALSE;
   BB2_SR2.Bef.Res_16 := FALSE;
   BB2_SR2.Bef.Res_17 := FALSE;
   BB2_SR2.Bef.Res_18 := FALSE;
   BB2_SR2.Bef.Res_19 := FALSE;
   BB2_SR2.Bef.Res_20 := FALSE;
   BB2_SR2.Bef.Res_21 := FALSE;
   BB2_SR2.Bef.Res_22 := FALSE;
   BB2_SR2.Bef.Res_23 := FALSE;
   BB2_SR2.Bef.Res_24 := FALSE;
   BB2_SR2.Bef.Res_25 := FALSE;
   BB2_SR2.Bef.Res_26 := FALSE;
   BB2_SR2.Bef.Res_27 := FALSE;
   BB2_SR2.Bef.Res_28 := FALSE;
   BB2_SR2.Bef.Res_29 := FALSE;
   BB2_SR2.Bef.BF_Set_SW_chg := FALSE;
   BB2_SR2.Bef.BF_Quit := FALSE;
   BB2_SR2.SW_Hand := 0.0;
   BB1_SR_K.Bef.Bed_Res := FALSE;
   BB1_SR_K.Bef.Bed_UV := FALSE;
   BB1_SR_K.Bef.Bed_NHV := FALSE;
   BB1_SR_K.Bef.Bed_PLS := FALSE;
   BB1_SR_K.Bef.BA_Hand := FALSE;
   BB1_SR_K.Bef.BA_Auto := FALSE;
   BB1_SR_K.Bef.BF_Ein1 := FALSE;
   BB1_SR_K.Bef.BF_Ein2 := FALSE;
   BB1_SR_K.Bef.BF_Aus := FALSE;
   BB1_SR_K.Bef.BZ_Res := FALSE;
   BB1_SR_K.Bef.Res_10 := FALSE;
   BB1_SR_K.Bef.Res_11 := FALSE;
   BB1_SR_K.Bef.Res_12 := FALSE;
   BB1_SR_K.Bef.Res_13 := FALSE;
   BB1_SR_K.Bef.Res_14 := FALSE;
   BB1_SR_K.Bef.Res_15 := FALSE;
   BB1_SR_K.Bef.Res_16 := FALSE;
   BB1_SR_K.Bef.Res_17 := FALSE;
   BB1_SR_K.Bef.Res_18 := FALSE;
   BB1_SR_K.Bef.Res_19 := FALSE;
   BB1_SR_K.Bef.Res_20 := FALSE;
   BB1_SR_K.Bef.Res_21 := FALSE;
   BB1_SR_K.Bef.Res_22 := FALSE;
   BB1_SR_K.Bef.Res_23 := FALSE;
   BB1_SR_K.Bef.Res_24 := FALSE;
   BB1_SR_K.Bef.Res_25 := FALSE;
   BB1_SR_K.Bef.Res_26 := FALSE;
   BB1_SR_K.Bef.Res_27 := FALSE;
   BB1_SR_K.Bef.Res_28 := FALSE;
   BB1_SR_K.Bef.Res_29 := FALSE;
   BB1_SR_K.Bef.BF_Set_SW_chg := FALSE;
   BB1_SR_K.Bef.BF_Quit := FALSE;
   BB1_SR_K.SW_Hand := 0.0;
   Zulauf_AR_P1.Bef.Bed_Res := FALSE;
   Zulauf_AR_P1.Bef.Bed_UV := FALSE;
   Zulauf_AR_P1.Bef.Bed_NHV := FALSE;
   Zulauf_AR_P1.Bef.Bed_PLS := FALSE;
   Zulauf_AR_P1.Bef.BA_Hand := FALSE;
   Zulauf_AR_P1.Bef.BA_Auto := FALSE;
   Zulauf_AR_P1.Bef.BF_Ein1 := FALSE;
   Zulauf_AR_P1.Bef.BF_Ein2 := FALSE;
   Zulauf_AR_P1.Bef.BF_Aus := FALSE;
   Zulauf_AR_P1.Bef.BZ_Res := FALSE;
   Zulauf_AR_P1.Bef.Res_10 := FALSE;
   Zulauf_AR_P1.Bef.Res_11 := FALSE;
   Zulauf_AR_P1.Bef.Res_12 := FALSE;
   Zulauf_AR_P1.Bef.Res_13 := FALSE;
   Zulauf_AR_P1.Bef.Res_14 := FALSE;
   Zulauf_AR_P1.Bef.Res_15 := FALSE;
   Zulauf_AR_P1.Bef.Res_16 := FALSE;
   Zulauf_AR_P1.Bef.Res_17 := FALSE;
   Zulauf_AR_P1.Bef.Res_18 := FALSE;
   Zulauf_AR_P1.Bef.Res_19 := FALSE;
   Zulauf_AR_P1.Bef.Res_20 := FALSE;
   Zulauf_AR_P1.Bef.Res_21 := FALSE;
   Zulauf_AR_P1.Bef.Res_22 := FALSE;
   Zulauf_AR_P1.Bef.Res_23 := FALSE;
   Zulauf_AR_P1.Bef.Res_24 := FALSE;
   Zulauf_AR_P1.Bef.Res_25 := FALSE;
   Zulauf_AR_P1.Bef.Res_26 := FALSE;
   Zulauf_AR_P1.Bef.Res_27 := FALSE;
   Zulauf_AR_P1.Bef.Res_28 := FALSE;
   Zulauf_AR_P1.Bef.Res_29 := FALSE;
   Zulauf_AR_P1.Bef.BF_Set_SW_chg := FALSE;
   Zulauf_AR_P1.Bef.BF_Quit := FALSE;
   Zulauf_AR_P1.SW_Hand := 0.0;
   Zulauf_AR_P2.Bef.Bed_Res := FALSE;
   Zulauf_AR_P2.Bef.Bed_UV := FALSE;
   Zulauf_AR_P2.Bef.Bed_NHV := FALSE;
   Zulauf_AR_P2.Bef.Bed_PLS := FALSE;
   Zulauf_AR_P2.Bef.BA_Hand := FALSE;
   Zulauf_AR_P2.Bef.BA_Auto := FALSE;
   Zulauf_AR_P2.Bef.BF_Ein1 := FALSE;
   Zulauf_AR_P2.Bef.BF_Ein2 := FALSE;
   Zulauf_AR_P2.Bef.BF_Aus := FALSE;
   Zulauf_AR_P2.Bef.BZ_Res := FALSE;
   Zulauf_AR_P2.Bef.Res_10 := FALSE;
   Zulauf_AR_P2.Bef.Res_11 := FALSE;
   Zulauf_AR_P2.Bef.Res_12 := FALSE;
   Zulauf_AR_P2.Bef.Res_13 := FALSE;
   Zulauf_AR_P2.Bef.Res_14 := FALSE;
   Zulauf_AR_P2.Bef.Res_15 := FALSE;
   Zulauf_AR_P2.Bef.Res_16 := FALSE;
   Zulauf_AR_P2.Bef.Res_17 := FALSE;
   Zulauf_AR_P2.Bef.Res_18 := FALSE;
   Zulauf_AR_P2.Bef.Res_19 := FALSE;
   Zulauf_AR_P2.Bef.Res_20 := FALSE;
   Zulauf_AR_P2.Bef.Res_21 := FALSE;
   Zulauf_AR_P2.Bef.Res_22 := FALSE;
   Zulauf_AR_P2.Bef.Res_23 := FALSE;
   Zulauf_AR_P2.Bef.Res_24 := FALSE;
   Zulauf_AR_P2.Bef.Res_25 := FALSE;
   Zulauf_AR_P2.Bef.Res_26 := FALSE;
   Zulauf_AR_P2.Bef.Res_27 := FALSE;
   Zulauf_AR_P2.Bef.Res_28 := FALSE;
   Zulauf_AR_P2.Bef.Res_29 := FALSE;
   Zulauf_AR_P2.Bef.BF_Set_SW_chg := FALSE;
   Zulauf_AR_P2.Bef.BF_Quit := FALSE;
   Zulauf_AR_P2.SW_Hand := 0.0;
   Zulauf_AS.Bef.Bed_Res := FALSE;
   Zulauf_AS.Bef.Bed_UV := FALSE;
   Zulauf_AS.Bef.Bed_NHV := FALSE;
   Zulauf_AS.Bef.Bed_PLS := FALSE;
   Zulauf_AS.Bef.BA_Hand := FALSE;
   Zulauf_AS.Bef.BA_Auto := FALSE;
   Zulauf_AS.Bef.BF_Ein1 := FALSE;
   Zulauf_AS.Bef.BF_Ein2 := FALSE;
   Zulauf_AS.Bef.BF_Aus := FALSE;
   Zulauf_AS.Bef.BZ_Res := FALSE;
   Zulauf_AS.Bef.Res_10 := FALSE;
   Zulauf_AS.Bef.Res_11 := FALSE;
   Zulauf_AS.Bef.Res_12 := FALSE;
   Zulauf_AS.Bef.Res_13 := FALSE;
   Zulauf_AS.Bef.Res_14 := FALSE;
   Zulauf_AS.Bef.Res_15 := FALSE;
   Zulauf_AS.Bef.Res_16 := FALSE;
   Zulauf_AS.Bef.Res_17 := FALSE;
   Zulauf_AS.Bef.Res_18 := FALSE;
   Zulauf_AS.Bef.Res_19 := FALSE;
   Zulauf_AS.Bef.Res_20 := FALSE;
   Zulauf_AS.Bef.Res_21 := FALSE;
   Zulauf_AS.Bef.Res_22 := FALSE;
   Zulauf_AS.Bef.Res_23 := FALSE;
   Zulauf_AS.Bef.Res_24 := FALSE;
   Zulauf_AS.Bef.Res_25 := FALSE;
   Zulauf_AS.Bef.Res_26 := FALSE;
   Zulauf_AS.Bef.Res_27 := FALSE;
   Zulauf_AS.Bef.Res_28 := FALSE;
   Zulauf_AS.Bef.Res_29 := FALSE;
   Zulauf_AS.Bef.BF_Set_SW_chg := FALSE;
   Zulauf_AS.Bef.BF_Quit := FALSE;
   Zulauf_AS.SW_Hand := 0.0;
   Zulauf_RA_SA.Bef.Bed_Res := FALSE;
   Zulauf_RA_SA.Bef.Bed_UV := FALSE;
   Zulauf_RA_SA.Bef.Bed_NHV := FALSE;
   Zulauf_RA_SA.Bef.Bed_PLS := FALSE;
   Zulauf_RA_SA.Bef.BA_Hand := FALSE;
   Zulauf_RA_SA.Bef.BA_Auto := FALSE;
   Zulauf_RA_SA.Bef.BF_Ein1 := FALSE;
   Zulauf_RA_SA.Bef.BF_Ein2 := FALSE;
   Zulauf_RA_SA.Bef.BF_Aus := FALSE;
   Zulauf_RA_SA.Bef.BZ_Res := FALSE;
   Zulauf_RA_SA.Bef.Res_10 := FALSE;
   Zulauf_RA_SA.Bef.Res_11 := FALSE;
   Zulauf_RA_SA.Bef.Res_12 := FALSE;
   Zulauf_RA_SA.Bef.Res_13 := FALSE;
   Zulauf_RA_SA.Bef.Res_14 := FALSE;
   Zulauf_RA_SA.Bef.Res_15 := FALSE;
   Zulauf_RA_SA.Bef.Res_16 := FALSE;
   Zulauf_RA_SA.Bef.Res_17 := FALSE;
   Zulauf_RA_SA.Bef.Res_18 := FALSE;
   Zulauf_RA_SA.Bef.Res_19 := FALSE;
   Zulauf_RA_SA.Bef.Res_20 := FALSE;
   Zulauf_RA_SA.Bef.Res_21 := FALSE;
   Zulauf_RA_SA.Bef.Res_22 := FALSE;
   Zulauf_RA_SA.Bef.Res_23 := FALSE;
   Zulauf_RA_SA.Bef.Res_24 := FALSE;
   Zulauf_RA_SA.Bef.Res_25 := FALSE;
   Zulauf_RA_SA.Bef.Res_26 := FALSE;
   Zulauf_RA_SA.Bef.Res_27 := FALSE;
   Zulauf_RA_SA.Bef.Res_28 := FALSE;
   Zulauf_RA_SA.Bef.Res_29 := FALSE;
   Zulauf_RA_SA.Bef.BF_Set_SW_chg := FALSE;
   Zulauf_RA_SA.Bef.BF_Quit := FALSE;
   Zulauf_RA_SA.SW_Hand := 0.0;
   Zulauf_RA_HZS.Bef.Bed_Res := FALSE;
   Zulauf_RA_HZS.Bef.Bed_UV := FALSE;
   Zulauf_RA_HZS.Bef.Bed_NHV := FALSE;
   Zulauf_RA_HZS.Bef.Bed_PLS := FALSE;
   Zulauf_RA_HZS.Bef.BA_Hand := FALSE;
   Zulauf_RA_HZS.Bef.BA_Auto := FALSE;
   Zulauf_RA_HZS.Bef.BF_Ein1 := FALSE;
   Zulauf_RA_HZS.Bef.BF_Ein2 := FALSE;
   Zulauf_RA_HZS.Bef.BF_Aus := FALSE;
   Zulauf_RA_HZS.Bef.BZ_Res := FALSE;
   Zulauf_RA_HZS.Bef.Res_10 := FALSE;
   Zulauf_RA_HZS.Bef.Res_11 := FALSE;
   Zulauf_RA_HZS.Bef.Res_12 := FALSE;
   Zulauf_RA_HZS.Bef.Res_13 := FALSE;
   Zulauf_RA_HZS.Bef.Res_14 := FALSE;
   Zulauf_RA_HZS.Bef.Res_15 := FALSE;
   Zulauf_RA_HZS.Bef.Res_16 := FALSE;
   Zulauf_RA_HZS.Bef.Res_17 := FALSE;
   Zulauf_RA_HZS.Bef.Res_18 := FALSE;
   Zulauf_RA_HZS.Bef.Res_19 := FALSE;
   Zulauf_RA_HZS.Bef.Res_20 := FALSE;
   Zulauf_RA_HZS.Bef.Res_21 := FALSE;
   Zulauf_RA_HZS.Bef.Res_22 := FALSE;
   Zulauf_RA_HZS.Bef.Res_23 := FALSE;
   Zulauf_RA_HZS.Bef.Res_24 := FALSE;
   Zulauf_RA_HZS.Bef.Res_25 := FALSE;
   Zulauf_RA_HZS.Bef.Res_26 := FALSE;
   Zulauf_RA_HZS.Bef.Res_27 := FALSE;
   Zulauf_RA_HZS.Bef.Res_28 := FALSE;
   Zulauf_RA_HZS.Bef.Res_29 := FALSE;
   Zulauf_RA_HZS.Bef.BF_Set_SW_chg := FALSE;
   Zulauf_RA_HZS.Bef.BF_Quit := FALSE;
   Zulauf_RA_HZS.SW_Hand := 0.0;
   Zulauf_RA_VKS.Bef.Bed_Res := FALSE;
   Zulauf_RA_VKS.Bef.Bed_UV := FALSE;
   Zulauf_RA_VKS.Bef.Bed_NHV := FALSE;
   Zulauf_RA_VKS.Bef.Bed_PLS := FALSE;
   Zulauf_RA_VKS.Bef.BA_Hand := FALSE;
   Zulauf_RA_VKS.Bef.BA_Auto := FALSE;
   Zulauf_RA_VKS.Bef.BF_Ein1 := FALSE;
   Zulauf_RA_VKS.Bef.BF_Ein2 := FALSE;
   Zulauf_RA_VKS.Bef.BF_Aus := FALSE;
   Zulauf_RA_VKS.Bef.BZ_Res := FALSE;
   Zulauf_RA_VKS.Bef.Res_10 := FALSE;
   Zulauf_RA_VKS.Bef.Res_11 := FALSE;
   Zulauf_RA_VKS.Bef.Res_12 := FALSE;
   Zulauf_RA_VKS.Bef.Res_13 := FALSE;
   Zulauf_RA_VKS.Bef.Res_14 := FALSE;
   Zulauf_RA_VKS.Bef.Res_15 := FALSE;
   Zulauf_RA_VKS.Bef.Res_16 := FALSE;
   Zulauf_RA_VKS.Bef.Res_17 := FALSE;
   Zulauf_RA_VKS.Bef.Res_18 := FALSE;
   Zulauf_RA_VKS.Bef.Res_19 := FALSE;
   Zulauf_RA_VKS.Bef.Res_20 := FALSE;
   Zulauf_RA_VKS.Bef.Res_21 := FALSE;
   Zulauf_RA_VKS.Bef.Res_22 := FALSE;
   Zulauf_RA_VKS.Bef.Res_23 := FALSE;
   Zulauf_RA_VKS.Bef.Res_24 := FALSE;
   Zulauf_RA_VKS.Bef.Res_25 := FALSE;
   Zulauf_RA_VKS.Bef.Res_26 := FALSE;
   Zulauf_RA_VKS.Bef.Res_27 := FALSE;
   Zulauf_RA_VKS.Bef.Res_28 := FALSE;
   Zulauf_RA_VKS.Bef.Res_29 := FALSE;
   Zulauf_RA_VKS.Bef.BF_Set_SW_chg := FALSE;
   Zulauf_RA_VKS.Bef.BF_Quit := FALSE;
   Zulauf_RA_VKS.SW_Hand := 0.0;
   Zulauf_RA_V.Bef.Bed_Res := FALSE;
   Zulauf_RA_V.Bef.Bed_UV := FALSE;
   Zulauf_RA_V.Bef.Bed_NHV := FALSE;
   Zulauf_RA_V.Bef.Bed_PLS := FALSE;
   Zulauf_RA_V.Bef.BA_Hand := FALSE;
   Zulauf_RA_V.Bef.BA_Auto := FALSE;
   Zulauf_RA_V.Bef.BF_Ein1 := FALSE;
   Zulauf_RA_V.Bef.BF_Ein2 := FALSE;
   Zulauf_RA_V.Bef.BF_Aus := FALSE;
   Zulauf_RA_V.Bef.BZ_Res := FALSE;
   Zulauf_RA_V.Bef.Res_10 := FALSE;
   Zulauf_RA_V.Bef.Res_11 := FALSE;
   Zulauf_RA_V.Bef.Res_12 := FALSE;
   Zulauf_RA_V.Bef.Res_13 := FALSE;
   Zulauf_RA_V.Bef.Res_14 := FALSE;
   Zulauf_RA_V.Bef.Res_15 := FALSE;
   Zulauf_RA_V.Bef.Res_16 := FALSE;
   Zulauf_RA_V.Bef.Res_17 := FALSE;
   Zulauf_RA_V.Bef.Res_18 := FALSE;
   Zulauf_RA_V.Bef.Res_19 := FALSE;
   Zulauf_RA_V.Bef.Res_20 := FALSE;
   Zulauf_RA_V.Bef.Res_21 := FALSE;
   Zulauf_RA_V.Bef.Res_22 := FALSE;
   Zulauf_RA_V.Bef.Res_23 := FALSE;
   Zulauf_RA_V.Bef.Res_24 := FALSE;
   Zulauf_RA_V.Bef.Res_25 := FALSE;
   Zulauf_RA_V.Bef.Res_26 := FALSE;
   Zulauf_RA_V.Bef.Res_27 := FALSE;
   Zulauf_RA_V.Bef.Res_28 := FALSE;
   Zulauf_RA_V.Bef.Res_29 := FALSE;
   Zulauf_RA_V.Bef.BF_Set_SW_chg := FALSE;
   Zulauf_RA_V.Bef.BF_Quit := FALSE;
   Zulauf_RA_V.SW_Hand := 0.0;
   Zulauf_RA_RP.Bef.Bed_Res := FALSE;
   Zulauf_RA_RP.Bef.Bed_UV := FALSE;
   Zulauf_RA_RP.Bef.Bed_NHV := FALSE;
   Zulauf_RA_RP.Bef.Bed_PLS := FALSE;
   Zulauf_RA_RP.Bef.BA_Hand := FALSE;
   Zulauf_RA_RP.Bef.BA_Auto := FALSE;
   Zulauf_RA_RP.Bef.BF_Ein1 := FALSE;
   Zulauf_RA_RP.Bef.BF_Ein2 := FALSE;
   Zulauf_RA_RP.Bef.BF_Aus := FALSE;
   Zulauf_RA_RP.Bef.BZ_Res := FALSE;
   Zulauf_RA_RP.Bef.Res_10 := FALSE;
   Zulauf_RA_RP.Bef.Res_11 := FALSE;
   Zulauf_RA_RP.Bef.Res_12 := FALSE;
   Zulauf_RA_RP.Bef.Res_13 := FALSE;
   Zulauf_RA_RP.Bef.Res_14 := FALSE;
   Zulauf_RA_RP.Bef.Res_15 := FALSE;
   Zulauf_RA_RP.Bef.Res_16 := FALSE;
   Zulauf_RA_RP.Bef.Res_17 := FALSE;
   Zulauf_RA_RP.Bef.Res_18 := FALSE;
   Zulauf_RA_RP.Bef.Res_19 := FALSE;
   Zulauf_RA_RP.Bef.Res_20 := FALSE;
   Zulauf_RA_RP.Bef.Res_21 := FALSE;
   Zulauf_RA_RP.Bef.Res_22 := FALSE;
   Zulauf_RA_RP.Bef.Res_23 := FALSE;
   Zulauf_RA_RP.Bef.Res_24 := FALSE;
   Zulauf_RA_RP.Bef.Res_25 := FALSE;
   Zulauf_RA_RP.Bef.Res_26 := FALSE;
   Zulauf_RA_RP.Bef.Res_27 := FALSE;
   Zulauf_RA_RP.Bef.Res_28 := FALSE;
   Zulauf_RA_RP.Bef.Res_29 := FALSE;
   Zulauf_RA_RP.Bef.BF_Set_SW_chg := FALSE;
   Zulauf_RA_RP.Bef.BF_Quit := FALSE;
   Zulauf_RA_RP.SW_Hand := 0.0;
   Zulauf_RA_FP.Bef.Bed_Res := FALSE;
   Zulauf_RA_FP.Bef.Bed_UV := FALSE;
   Zulauf_RA_FP.Bef.Bed_NHV := FALSE;
   Zulauf_RA_FP.Bef.Bed_PLS := FALSE;
   Zulauf_RA_FP.Bef.BA_Hand := FALSE;
   Zulauf_RA_FP.Bef.BA_Auto := FALSE;
   Zulauf_RA_FP.Bef.BF_Ein1 := FALSE;
   Zulauf_RA_FP.Bef.BF_Ein2 := FALSE;
   Zulauf_RA_FP.Bef.BF_Aus := FALSE;
   Zulauf_RA_FP.Bef.BZ_Res := FALSE;
   Zulauf_RA_FP.Bef.Res_10 := FALSE;
   Zulauf_RA_FP.Bef.Res_11 := FALSE;
   Zulauf_RA_FP.Bef.Res_12 := FALSE;
   Zulauf_RA_FP.Bef.Res_13 := FALSE;
   Zulauf_RA_FP.Bef.Res_14 := FALSE;
   Zulauf_RA_FP.Bef.Res_15 := FALSE;
   Zulauf_RA_FP.Bef.Res_16 := FALSE;
   Zulauf_RA_FP.Bef.Res_17 := FALSE;
   Zulauf_RA_FP.Bef.Res_18 := FALSE;
   Zulauf_RA_FP.Bef.Res_19 := FALSE;
   Zulauf_RA_FP.Bef.Res_20 := FALSE;
   Zulauf_RA_FP.Bef.Res_21 := FALSE;
   Zulauf_RA_FP.Bef.Res_22 := FALSE;
   Zulauf_RA_FP.Bef.Res_23 := FALSE;
   Zulauf_RA_FP.Bef.Res_24 := FALSE;
   Zulauf_RA_FP.Bef.Res_25 := FALSE;
   Zulauf_RA_FP.Bef.Res_26 := FALSE;
   Zulauf_RA_FP.Bef.Res_27 := FALSE;
   Zulauf_RA_FP.Bef.Res_28 := FALSE;
   Zulauf_RA_FP.Bef.Res_29 := FALSE;
   Zulauf_RA_FP.Bef.BF_Set_SW_chg := FALSE;
   Zulauf_RA_FP.Bef.BF_Quit := FALSE;
   Zulauf_RA_FP.SW_Hand := 0.0;
   Schlamm_BP.Bef.Bed_Res := FALSE;
   Schlamm_BP.Bef.Bed_UV := FALSE;
   Schlamm_BP.Bef.Bed_NHV := FALSE;
   Schlamm_BP.Bef.Bed_PLS := FALSE;
   Schlamm_BP.Bef.BA_Hand := FALSE;
   Schlamm_BP.Bef.BA_Auto := FALSE;
   Schlamm_BP.Bef.BF_Ein1 := FALSE;
   Schlamm_BP.Bef.BF_Ein2 := FALSE;
   Schlamm_BP.Bef.BF_Aus := FALSE;
   Schlamm_BP.Bef.BZ_Res := FALSE;
   Schlamm_BP.Bef.Res_10 := FALSE;
   Schlamm_BP.Bef.Res_11 := FALSE;
   Schlamm_BP.Bef.Res_12 := FALSE;
   Schlamm_BP.Bef.Res_13 := FALSE;
   Schlamm_BP.Bef.Res_14 := FALSE;
   Schlamm_BP.Bef.Res_15 := FALSE;
   Schlamm_BP.Bef.Res_16 := FALSE;
   Schlamm_BP.Bef.Res_17 := FALSE;
   Schlamm_BP.Bef.Res_18 := FALSE;
   Schlamm_BP.Bef.Res_19 := FALSE;
   Schlamm_BP.Bef.Res_20 := FALSE;
   Schlamm_BP.Bef.Res_21 := FALSE;
   Schlamm_BP.Bef.Res_22 := FALSE;
   Schlamm_BP.Bef.Res_23 := FALSE;
   Schlamm_BP.Bef.Res_24 := FALSE;
   Schlamm_BP.Bef.Res_25 := FALSE;
   Schlamm_BP.Bef.Res_26 := FALSE;
   Schlamm_BP.Bef.Res_27 := FALSE;
   Schlamm_BP.Bef.Res_28 := FALSE;
   Schlamm_BP.Bef.Res_29 := FALSE;
   Schlamm_BP.Bef.BF_Set_SW_chg := FALSE;
   Schlamm_BP.Bef.BF_Quit := FALSE;
   Schlamm_BP.SW_Hand := 0.0;
   Truebwasser_P1.Bef.Bed_Res := FALSE;
   Truebwasser_P1.Bef.Bed_UV := FALSE;
   Truebwasser_P1.Bef.Bed_NHV := FALSE;
   Truebwasser_P1.Bef.Bed_PLS := FALSE;
   Truebwasser_P1.Bef.BA_Hand := FALSE;
   Truebwasser_P1.Bef.BA_Auto := FALSE;
   Truebwasser_P1.Bef.BF_Ein1 := FALSE;
   Truebwasser_P1.Bef.BF_Ein2 := FALSE;
   Truebwasser_P1.Bef.BF_Aus := FALSE;
   Truebwasser_P1.Bef.BZ_Res := FALSE;
   Truebwasser_P1.Bef.Res_10 := FALSE;
   Truebwasser_P1.Bef.Res_11 := FALSE;
   Truebwasser_P1.Bef.Res_12 := FALSE;
   Truebwasser_P1.Bef.Res_13 := FALSE;
   Truebwasser_P1.Bef.Res_14 := FALSE;
   Truebwasser_P1.Bef.Res_15 := FALSE;
   Truebwasser_P1.Bef.Res_16 := FALSE;
   Truebwasser_P1.Bef.Res_17 := FALSE;
   Truebwasser_P1.Bef.Res_18 := FALSE;
   Truebwasser_P1.Bef.Res_19 := FALSE;
   Truebwasser_P1.Bef.Res_20 := FALSE;
   Truebwasser_P1.Bef.Res_21 := FALSE;
   Truebwasser_P1.Bef.Res_22 := FALSE;
   Truebwasser_P1.Bef.Res_23 := FALSE;
   Truebwasser_P1.Bef.Res_24 := FALSE;
   Truebwasser_P1.Bef.Res_25 := FALSE;
   Truebwasser_P1.Bef.Res_26 := FALSE;
   Truebwasser_P1.Bef.Res_27 := FALSE;
   Truebwasser_P1.Bef.Res_28 := FALSE;
   Truebwasser_P1.Bef.Res_29 := FALSE;
   Truebwasser_P1.Bef.BF_Set_SW_chg := FALSE;
   Truebwasser_P1.Bef.BF_Quit := FALSE;
   Truebwasser_P1.SW_Hand := 0.0;
   Truebwasser_P2.Bef.Bed_Res := FALSE;
   Truebwasser_P2.Bef.Bed_UV := FALSE;
   Truebwasser_P2.Bef.Bed_NHV := FALSE;
   Truebwasser_P2.Bef.Bed_PLS := FALSE;
   Truebwasser_P2.Bef.BA_Hand := FALSE;
   Truebwasser_P2.Bef.BA_Auto := FALSE;
   Truebwasser_P2.Bef.BF_Ein1 := FALSE;
   Truebwasser_P2.Bef.BF_Ein2 := FALSE;
   Truebwasser_P2.Bef.BF_Aus := FALSE;
   Truebwasser_P2.Bef.BZ_Res := FALSE;
   Truebwasser_P2.Bef.Res_10 := FALSE;
   Truebwasser_P2.Bef.Res_11 := FALSE;
   Truebwasser_P2.Bef.Res_12 := FALSE;
   Truebwasser_P2.Bef.Res_13 := FALSE;
   Truebwasser_P2.Bef.Res_14 := FALSE;
   Truebwasser_P2.Bef.Res_15 := FALSE;
   Truebwasser_P2.Bef.Res_16 := FALSE;
   Truebwasser_P2.Bef.Res_17 := FALSE;
   Truebwasser_P2.Bef.Res_18 := FALSE;
   Truebwasser_P2.Bef.Res_19 := FALSE;
   Truebwasser_P2.Bef.Res_20 := FALSE;
   Truebwasser_P2.Bef.Res_21 := FALSE;
   Truebwasser_P2.Bef.Res_22 := FALSE;
   Truebwasser_P2.Bef.Res_23 := FALSE;
   Truebwasser_P2.Bef.Res_24 := FALSE;
   Truebwasser_P2.Bef.Res_25 := FALSE;
   Truebwasser_P2.Bef.Res_26 := FALSE;
   Truebwasser_P2.Bef.Res_27 := FALSE;
   Truebwasser_P2.Bef.Res_28 := FALSE;
   Truebwasser_P2.Bef.Res_29 := FALSE;
   Truebwasser_P2.Bef.BF_Set_SW_chg := FALSE;
   Truebwasser_P2.Bef.BF_Quit := FALSE;
   Truebwasser_P2.SW_Hand := 0.0;
   Schlamm_AS.Bef.Bed_Res := FALSE;
   Schlamm_AS.Bef.Bed_UV := FALSE;
   Schlamm_AS.Bef.Bed_NHV := FALSE;
   Schlamm_AS.Bef.Bed_PLS := FALSE;
   Schlamm_AS.Bef.BA_Hand := FALSE;
   Schlamm_AS.Bef.BA_Auto := FALSE;
   Schlamm_AS.Bef.BF_Ein1 := FALSE;
   Schlamm_AS.Bef.BF_Ein2 := FALSE;
   Schlamm_AS.Bef.BF_Aus := FALSE;
   Schlamm_AS.Bef.BZ_Res := FALSE;
   Schlamm_AS.Bef.Res_10 := FALSE;
   Schlamm_AS.Bef.Res_11 := FALSE;
   Schlamm_AS.Bef.Res_12 := FALSE;
   Schlamm_AS.Bef.Res_13 := FALSE;
   Schlamm_AS.Bef.Res_14 := FALSE;
   Schlamm_AS.Bef.Res_15 := FALSE;
   Schlamm_AS.Bef.Res_16 := FALSE;
   Schlamm_AS.Bef.Res_17 := FALSE;
   Schlamm_AS.Bef.Res_18 := FALSE;
   Schlamm_AS.Bef.Res_19 := FALSE;
   Schlamm_AS.Bef.Res_20 := FALSE;
   Schlamm_AS.Bef.Res_21 := FALSE;
   Schlamm_AS.Bef.Res_22 := FALSE;
   Schlamm_AS.Bef.Res_23 := FALSE;
   Schlamm_AS.Bef.Res_24 := FALSE;
   Schlamm_AS.Bef.Res_25 := FALSE;
   Schlamm_AS.Bef.Res_26 := FALSE;
   Schlamm_AS.Bef.Res_27 := FALSE;
   Schlamm_AS.Bef.Res_28 := FALSE;
   Schlamm_AS.Bef.Res_29 := FALSE;
   Schlamm_AS.Bef.BF_Set_SW_chg := FALSE;
   Schlamm_AS.Bef.BF_Quit := FALSE;
   Schlamm_AS.SW_Hand := 0.0;
   BB2_SR_K.Bef.Bed_Res := FALSE;
   BB2_SR_K.Bef.Bed_UV := FALSE;
   BB2_SR_K.Bef.Bed_NHV := FALSE;
   BB2_SR_K.Bef.Bed_PLS := FALSE;
   BB2_SR_K.Bef.BA_Hand := FALSE;
   BB2_SR_K.Bef.BA_Auto := FALSE;
   BB2_SR_K.Bef.BF_Ein1 := FALSE;
   BB2_SR_K.Bef.BF_Ein2 := FALSE;
   BB2_SR_K.Bef.BF_Aus := FALSE;
   BB2_SR_K.Bef.BZ_Res := FALSE;
   BB2_SR_K.Bef.Res_10 := FALSE;
   BB2_SR_K.Bef.Res_11 := FALSE;
   BB2_SR_K.Bef.Res_12 := FALSE;
   BB2_SR_K.Bef.Res_13 := FALSE;
   BB2_SR_K.Bef.Res_14 := FALSE;
   BB2_SR_K.Bef.Res_15 := FALSE;
   BB2_SR_K.Bef.Res_16 := FALSE;
   BB2_SR_K.Bef.Res_17 := FALSE;
   BB2_SR_K.Bef.Res_18 := FALSE;
   BB2_SR_K.Bef.Res_19 := FALSE;
   BB2_SR_K.Bef.Res_20 := FALSE;
   BB2_SR_K.Bef.Res_21 := FALSE;
   BB2_SR_K.Bef.Res_22 := FALSE;
   BB2_SR_K.Bef.Res_23 := FALSE;
   BB2_SR_K.Bef.Res_24 := FALSE;
   BB2_SR_K.Bef.Res_25 := FALSE;
   BB2_SR_K.Bef.Res_26 := FALSE;
   BB2_SR_K.Bef.Res_27 := FALSE;
   BB2_SR_K.Bef.Res_28 := FALSE;
   BB2_SR_K.Bef.Res_29 := FALSE;
   BB2_SR_K.Bef.BF_Set_SW_chg := FALSE;
   BB2_SR_K.Bef.BF_Quit := FALSE;
   BB2_SR_K.SW_Hand := 0.0;

END_DATA_BLOCK

DATA_BLOCK "DB91_DP_aktiv"
{ S7_Optimized_Access := 'TRUE' }
VERSION : 0.1
NON_RETAIN
   VAR
      Tln : Array[0..127] of Bool;
   END_VAR


BEGIN
   Tln[0] := TRUE;
   Tln[1] := FALSE;
   Tln[2] := FALSE;
   Tln[3] := TRUE;
   Tln[4] := TRUE;
   Tln[5] := TRUE;
   Tln[6] := TRUE;
   Tln[7] := TRUE;
   Tln[8] := FALSE;
   Tln[9] := FALSE;
   Tln[10] := TRUE;
   Tln[11] := TRUE;
   Tln[12] := FALSE;
   Tln[13] := FALSE;
   Tln[14] := FALSE;
   Tln[15] := FALSE;
   Tln[16] := FALSE;
   Tln[17] := FALSE;
   Tln[18] := FALSE;
   Tln[19] := FALSE;
   Tln[20] := FALSE;
   Tln[21] := FALSE;
   Tln[22] := FALSE;
   Tln[23] := FALSE;
   Tln[24] := FALSE;
   Tln[25] := FALSE;
   Tln[26] := FALSE;
   Tln[27] := FALSE;
   Tln[28] := FALSE;
   Tln[29] := FALSE;
   Tln[30] := FALSE;
   Tln[31] := FALSE;
   Tln[32] := FALSE;
   Tln[33] := FALSE;
   Tln[34] := FALSE;
   Tln[35] := FALSE;
   Tln[36] := FALSE;
   Tln[37] := FALSE;
   Tln[38] := FALSE;
   Tln[39] := FALSE;
   Tln[40] := FALSE;
   Tln[41] := FALSE;
   Tln[42] := FALSE;
   Tln[43] := FALSE;
   Tln[44] := FALSE;
   Tln[45] := FALSE;
   Tln[46] := FALSE;
   Tln[47] := FALSE;
   Tln[48] := FALSE;
   Tln[49] := FALSE;
   Tln[50] := FALSE;
   Tln[51] := FALSE;
   Tln[52] := FALSE;
   Tln[53] := FALSE;
   Tln[54] := FALSE;
   Tln[55] := FALSE;
   Tln[56] := FALSE;
   Tln[57] := FALSE;
   Tln[58] := FALSE;
   Tln[59] := FALSE;
   Tln[60] := FALSE;
   Tln[61] := FALSE;
   Tln[62] := FALSE;
   Tln[63] := FALSE;
   Tln[64] := FALSE;
   Tln[65] := FALSE;
   Tln[66] := FALSE;
   Tln[67] := FALSE;
   Tln[68] := FALSE;
   Tln[69] := FALSE;
   Tln[70] := FALSE;
   Tln[71] := FALSE;
   Tln[72] := FALSE;
   Tln[73] := FALSE;
   Tln[74] := FALSE;
   Tln[75] := FALSE;
   Tln[76] := FALSE;
   Tln[77] := FALSE;
   Tln[78] := FALSE;
   Tln[79] := FALSE;
   Tln[80] := FALSE;
   Tln[81] := FALSE;
   Tln[82] := FALSE;
   Tln[83] := FALSE;
   Tln[84] := FALSE;
   Tln[85] := FALSE;
   Tln[86] := FALSE;
   Tln[87] := FALSE;
   Tln[88] := FALSE;
   Tln[89] := FALSE;
   Tln[90] := FALSE;
   Tln[91] := FALSE;
   Tln[92] := FALSE;
   Tln[93] := FALSE;
   Tln[94] := FALSE;
   Tln[95] := FALSE;
   Tln[96] := FALSE;
   Tln[97] := FALSE;
   Tln[98] := FALSE;
   Tln[99] := FALSE;
   Tln[100] := FALSE;
   Tln[101] := FALSE;
   Tln[102] := FALSE;
   Tln[103] := FALSE;
   Tln[104] := FALSE;
   Tln[105] := FALSE;
   Tln[106] := FALSE;
   Tln[107] := FALSE;
   Tln[108] := FALSE;
   Tln[109] := FALSE;
   Tln[110] := FALSE;
   Tln[111] := FALSE;
   Tln[112] := FALSE;
   Tln[113] := FALSE;
   Tln[114] := FALSE;
   Tln[115] := FALSE;
   Tln[116] := FALSE;
   Tln[117] := FALSE;
   Tln[118] := FALSE;
   Tln[119] := FALSE;
   Tln[120] := FALSE;
   Tln[121] := FALSE;
   Tln[122] := FALSE;
   Tln[123] := FALSE;
   Tln[124] := FALSE;
   Tln[125] := FALSE;
   Tln[126] := FALSE;
   Tln[127] := FALSE;

END_DATA_BLOCK

DATA_BLOCK "DB105_Antriebe_Bef_PLS"
{ S7_Optimized_Access := 'FALSE' }
VERSION : 0.1
NON_RETAIN
   STRUCT
      BB_G1 : "T_ANTRIEB_BEF";   // Belebung - Gebläse 1
      BB_G2 : "T_ANTRIEB_BEF";   // Belebung - Gebläse 2
      BB_G3 : "T_ANTRIEB_BEF";   // Belebung - Gebläse 3
      BB_SHL_G1 : "T_ANTRIEB_BEF";   // Belebung - Schallhaubenlüfter Gebläse 1
      BB_SHL_G2 : "T_ANTRIEB_BEF";   // Belebung - Schallhaubenlüfter Gebläse 2
      BB_SHL_G3 : "T_ANTRIEB_BEF";   // Belebung - Schallhaubenlüfter Gebläse 3
      BB_AV : "T_ANTRIEB_BEF";   // Belebung - Gebläsestation - Abluftventilator
      BB_LS1 : "T_ANTRIEB_BEF";   // Belebung - Gebläsestation - Luftwegschieber 1
      BB_LS2 : "T_ANTRIEB_BEF";   // Belebung - Gebläsestation - Luftwegschieber 2
      BB1_RZP1 : "T_ANTRIEB_BEF";   // Becken 1 - Rezipumpe 1
      BB1_RZP2 : "T_ANTRIEB_BEF";   // Becken 1 - Rezipumpe 2
      BB1_UeSP : "T_ANTRIEB_BEF";   // Becken 1 - ÜSS-Pumpe
      BB1_AS1 : "T_ANTRIEB_BEF";   // Becken 1 - Ablaufschieber 1
      BB1_AS2 : "T_ANTRIEB_BEF";   // Becken 1 - Ablaufschieber 2
      BB1_SR1 : "T_ANTRIEB_BEF";   // Becken 1 - MV Schlammrückführung 1
      BB1_SR2 : "T_ANTRIEB_BEF";   // Becken 1 - MV Schlammrückführung 2
      BB2_RZP1 : "T_ANTRIEB_BEF";   // Becken 2 - Rezipumpe 1
      BB2_RZP2 : "T_ANTRIEB_BEF";   // Becken 2 - Rezipumpe 2
      BB2_UeSP : "T_ANTRIEB_BEF";   // Becken 2 - ÜSS-Pumpe
      BB2_AS1 : "T_ANTRIEB_BEF";   // Becken 2 - Ablaufschieber 1
      BB2_AS2 : "T_ANTRIEB_BEF";   // Becken 2 - Ablaufschieber 2
      BB2_SR1 : "T_ANTRIEB_BEF";   // Becken 2 - MV Schlammrückführung 1
      BB2_SR2 : "T_ANTRIEB_BEF";   // Becken 2 - MV Schlammrückführung 2
      BB1_SR_K : "T_ANTRIEB_BEF";   // Becken 1- Druckluftkompressor Schlammrückführung
      Zulauf_AR_P1 : "T_ANTRIEB_BEF";   // Zulauf - Pumpwerk "Alter Rechen" - Pumpe 1
      Zulauf_AR_P2 : "T_ANTRIEB_BEF";   // Zulauf - Pumpwerk "Alter Rechen" - Pumpe 2
      Zulauf_AS : "T_ANTRIEB_BEF";   // Zulauf - Vorlagebehälter - Absperrschieber
      Zulauf_RA_SA : "T_ANTRIEB_BEF";   // Zulauf - Rechen - Sieb
      Zulauf_RA_HZS : "T_ANTRIEB_BEF";   // Zulauf - Rechen - HZS
      Zulauf_RA_VKS : "T_ANTRIEB_BEF";   // Zulauf - Rechen - VZS
      Zulauf_RA_V : "T_ANTRIEB_BEF";   // Zulauf - Rechen - Belüfter
      Zulauf_RA_RP : "T_ANTRIEB_BEF";   // Zulauf - Rechen - Räumpaddel
      Zulauf_RA_FP : "T_ANTRIEB_BEF";   // Zulauf - Rechen - Fettpumpe
      Schlamm_BP : "T_ANTRIEB_BEF";   // Schlamm - Beschickungspumpe Schlammbeete
      Truebwasser_P1 : "T_ANTRIEB_BEF";   // Trübwasserpumpwerk - Pumpe 1
      Truebwasser_P2 : "T_ANTRIEB_BEF";   // Trübwasserpumpwerk - Pumpe 2
      Schlamm_AS : "T_ANTRIEB_BEF";   // Schlamm - Absperrschieber Schlammbeete
      BB2_SR_K : "T_ANTRIEB_BEF";   // Becken 2 - Druckluftkompressor Schlammrückführung
      Zulauf_DosP : "T_ANTRIEB_BEF";   // Zulauf - Dosierpumpe
   END_STRUCT;


BEGIN
   BB_G1.Bef.Bed_Res := FALSE;
   BB_G1.Bef.Bed_UV := FALSE;
   BB_G1.Bef.Bed_NHV := FALSE;
   BB_G1.Bef.Bed_PLS := FALSE;
   BB_G1.Bef.BA_Hand := FALSE;
   BB_G1.Bef.BA_Auto := FALSE;
   BB_G1.Bef.BF_Ein1 := FALSE;
   BB_G1.Bef.BF_Ein2 := FALSE;
   BB_G1.Bef.BF_Aus := FALSE;
   BB_G1.Bef.BZ_Res := FALSE;
   BB_G1.Bef.Res_10 := FALSE;
   BB_G1.Bef.Res_11 := FALSE;
   BB_G1.Bef.Res_12 := FALSE;
   BB_G1.Bef.Res_13 := FALSE;
   BB_G1.Bef.Res_14 := FALSE;
   BB_G1.Bef.Res_15 := FALSE;
   BB_G1.Bef.Res_16 := FALSE;
   BB_G1.Bef.Res_17 := FALSE;
   BB_G1.Bef.Res_18 := FALSE;
   BB_G1.Bef.Res_19 := FALSE;
   BB_G1.Bef.Res_20 := FALSE;
   BB_G1.Bef.Res_21 := FALSE;
   BB_G1.Bef.Res_22 := FALSE;
   BB_G1.Bef.Res_23 := FALSE;
   BB_G1.Bef.Res_24 := FALSE;
   BB_G1.Bef.Res_25 := FALSE;
   BB_G1.Bef.Res_26 := FALSE;
   BB_G1.Bef.Res_27 := FALSE;
   BB_G1.Bef.Res_28 := FALSE;
   BB_G1.Bef.Res_29 := FALSE;
   BB_G1.Bef.BF_Set_SW_chg := FALSE;
   BB_G1.Bef.BF_Quit := FALSE;
   BB_G1.SW_Hand := 0.0;
   BB_G2.Bef.Bed_Res := FALSE;
   BB_G2.Bef.Bed_UV := FALSE;
   BB_G2.Bef.Bed_NHV := FALSE;
   BB_G2.Bef.Bed_PLS := FALSE;
   BB_G2.Bef.BA_Hand := FALSE;
   BB_G2.Bef.BA_Auto := FALSE;
   BB_G2.Bef.BF_Ein1 := FALSE;
   BB_G2.Bef.BF_Ein2 := FALSE;
   BB_G2.Bef.BF_Aus := FALSE;
   BB_G2.Bef.BZ_Res := FALSE;
   BB_G2.Bef.Res_10 := FALSE;
   BB_G2.Bef.Res_11 := FALSE;
   BB_G2.Bef.Res_12 := FALSE;
   BB_G2.Bef.Res_13 := FALSE;
   BB_G2.Bef.Res_14 := FALSE;
   BB_G2.Bef.Res_15 := FALSE;
   BB_G2.Bef.Res_16 := FALSE;
   BB_G2.Bef.Res_17 := FALSE;
   BB_G2.Bef.Res_18 := FALSE;
   BB_G2.Bef.Res_19 := FALSE;
   BB_G2.Bef.Res_20 := FALSE;
   BB_G2.Bef.Res_21 := FALSE;
   BB_G2.Bef.Res_22 := FALSE;
   BB_G2.Bef.Res_23 := FALSE;
   BB_G2.Bef.Res_24 := FALSE;
   BB_G2.Bef.Res_25 := FALSE;
   BB_G2.Bef.Res_26 := FALSE;
   BB_G2.Bef.Res_27 := FALSE;
   BB_G2.Bef.Res_28 := FALSE;
   BB_G2.Bef.Res_29 := FALSE;
   BB_G2.Bef.BF_Set_SW_chg := FALSE;
   BB_G2.Bef.BF_Quit := FALSE;
   BB_G2.SW_Hand := 0.0;
   BB_G3.Bef.Bed_Res := FALSE;
   BB_G3.Bef.Bed_UV := FALSE;
   BB_G3.Bef.Bed_NHV := FALSE;
   BB_G3.Bef.Bed_PLS := FALSE;
   BB_G3.Bef.BA_Hand := FALSE;
   BB_G3.Bef.BA_Auto := FALSE;
   BB_G3.Bef.BF_Ein1 := FALSE;
   BB_G3.Bef.BF_Ein2 := FALSE;
   BB_G3.Bef.BF_Aus := FALSE;
   BB_G3.Bef.BZ_Res := FALSE;
   BB_G3.Bef.Res_10 := FALSE;
   BB_G3.Bef.Res_11 := FALSE;
   BB_G3.Bef.Res_12 := FALSE;
   BB_G3.Bef.Res_13 := FALSE;
   BB_G3.Bef.Res_14 := FALSE;
   BB_G3.Bef.Res_15 := FALSE;
   BB_G3.Bef.Res_16 := FALSE;
   BB_G3.Bef.Res_17 := FALSE;
   BB_G3.Bef.Res_18 := FALSE;
   BB_G3.Bef.Res_19 := FALSE;
   BB_G3.Bef.Res_20 := FALSE;
   BB_G3.Bef.Res_21 := FALSE;
   BB_G3.Bef.Res_22 := FALSE;
   BB_G3.Bef.Res_23 := FALSE;
   BB_G3.Bef.Res_24 := FALSE;
   BB_G3.Bef.Res_25 := FALSE;
   BB_G3.Bef.Res_26 := FALSE;
   BB_G3.Bef.Res_27 := FALSE;
   BB_G3.Bef.Res_28 := FALSE;
   BB_G3.Bef.Res_29 := FALSE;
   BB_G3.Bef.BF_Set_SW_chg := FALSE;
   BB_G3.Bef.BF_Quit := FALSE;
   BB_G3.SW_Hand := 0.0;
   BB_SHL_G1.Bef.Bed_Res := FALSE;
   BB_SHL_G1.Bef.Bed_UV := FALSE;
   BB_SHL_G1.Bef.Bed_NHV := FALSE;
   BB_SHL_G1.Bef.Bed_PLS := FALSE;
   BB_SHL_G1.Bef.BA_Hand := FALSE;
   BB_SHL_G1.Bef.BA_Auto := FALSE;
   BB_SHL_G1.Bef.BF_Ein1 := FALSE;
   BB_SHL_G1.Bef.BF_Ein2 := FALSE;
   BB_SHL_G1.Bef.BF_Aus := FALSE;
   BB_SHL_G1.Bef.BZ_Res := FALSE;
   BB_SHL_G1.Bef.Res_10 := FALSE;
   BB_SHL_G1.Bef.Res_11 := FALSE;
   BB_SHL_G1.Bef.Res_12 := FALSE;
   BB_SHL_G1.Bef.Res_13 := FALSE;
   BB_SHL_G1.Bef.Res_14 := FALSE;
   BB_SHL_G1.Bef.Res_15 := FALSE;
   BB_SHL_G1.Bef.Res_16 := FALSE;
   BB_SHL_G1.Bef.Res_17 := FALSE;
   BB_SHL_G1.Bef.Res_18 := FALSE;
   BB_SHL_G1.Bef.Res_19 := FALSE;
   BB_SHL_G1.Bef.Res_20 := FALSE;
   BB_SHL_G1.Bef.Res_21 := FALSE;
   BB_SHL_G1.Bef.Res_22 := FALSE;
   BB_SHL_G1.Bef.Res_23 := FALSE;
   BB_SHL_G1.Bef.Res_24 := FALSE;
   BB_SHL_G1.Bef.Res_25 := FALSE;
   BB_SHL_G1.Bef.Res_26 := FALSE;
   BB_SHL_G1.Bef.Res_27 := FALSE;
   BB_SHL_G1.Bef.Res_28 := FALSE;
   BB_SHL_G1.Bef.Res_29 := FALSE;
   BB_SHL_G1.Bef.BF_Set_SW_chg := FALSE;
   BB_SHL_G1.Bef.BF_Quit := FALSE;
   BB_SHL_G1.SW_Hand := 0.0;
   BB_SHL_G2.Bef.Bed_Res := FALSE;
   BB_SHL_G2.Bef.Bed_UV := FALSE;
   BB_SHL_G2.Bef.Bed_NHV := FALSE;
   BB_SHL_G2.Bef.Bed_PLS := FALSE;
   BB_SHL_G2.Bef.BA_Hand := FALSE;
   BB_SHL_G2.Bef.BA_Auto := FALSE;
   BB_SHL_G2.Bef.BF_Ein1 := FALSE;
   BB_SHL_G2.Bef.BF_Ein2 := FALSE;
   BB_SHL_G2.Bef.BF_Aus := FALSE;
   BB_SHL_G2.Bef.BZ_Res := FALSE;
   BB_SHL_G2.Bef.Res_10 := FALSE;
   BB_SHL_G2.Bef.Res_11 := FALSE;
   BB_SHL_G2.Bef.Res_12 := FALSE;
   BB_SHL_G2.Bef.Res_13 := FALSE;
   BB_SHL_G2.Bef.Res_14 := FALSE;
   BB_SHL_G2.Bef.Res_15 := FALSE;
   BB_SHL_G2.Bef.Res_16 := FALSE;
   BB_SHL_G2.Bef.Res_17 := FALSE;
   BB_SHL_G2.Bef.Res_18 := FALSE;
   BB_SHL_G2.Bef.Res_19 := FALSE;
   BB_SHL_G2.Bef.Res_20 := FALSE;
   BB_SHL_G2.Bef.Res_21 := FALSE;
   BB_SHL_G2.Bef.Res_22 := FALSE;
   BB_SHL_G2.Bef.Res_23 := FALSE;
   BB_SHL_G2.Bef.Res_24 := FALSE;
   BB_SHL_G2.Bef.Res_25 := FALSE;
   BB_SHL_G2.Bef.Res_26 := FALSE;
   BB_SHL_G2.Bef.Res_27 := FALSE;
   BB_SHL_G2.Bef.Res_28 := FALSE;
   BB_SHL_G2.Bef.Res_29 := FALSE;
   BB_SHL_G2.Bef.BF_Set_SW_chg := FALSE;
   BB_SHL_G2.Bef.BF_Quit := FALSE;
   BB_SHL_G2.SW_Hand := 0.0;
   BB_SHL_G3.Bef.Bed_Res := FALSE;
   BB_SHL_G3.Bef.Bed_UV := FALSE;
   BB_SHL_G3.Bef.Bed_NHV := FALSE;
   BB_SHL_G3.Bef.Bed_PLS := FALSE;
   BB_SHL_G3.Bef.BA_Hand := FALSE;
   BB_SHL_G3.Bef.BA_Auto := FALSE;
   BB_SHL_G3.Bef.BF_Ein1 := FALSE;
   BB_SHL_G3.Bef.BF_Ein2 := FALSE;
   BB_SHL_G3.Bef.BF_Aus := FALSE;
   BB_SHL_G3.Bef.BZ_Res := FALSE;
   BB_SHL_G3.Bef.Res_10 := FALSE;
   BB_SHL_G3.Bef.Res_11 := FALSE;
   BB_SHL_G3.Bef.Res_12 := FALSE;
   BB_SHL_G3.Bef.Res_13 := FALSE;
   BB_SHL_G3.Bef.Res_14 := FALSE;
   BB_SHL_G3.Bef.Res_15 := FALSE;
   BB_SHL_G3.Bef.Res_16 := FALSE;
   BB_SHL_G3.Bef.Res_17 := FALSE;
   BB_SHL_G3.Bef.Res_18 := FALSE;
   BB_SHL_G3.Bef.Res_19 := FALSE;
   BB_SHL_G3.Bef.Res_20 := FALSE;
   BB_SHL_G3.Bef.Res_21 := FALSE;
   BB_SHL_G3.Bef.Res_22 := FALSE;
   BB_SHL_G3.Bef.Res_23 := FALSE;
   BB_SHL_G3.Bef.Res_24 := FALSE;
   BB_SHL_G3.Bef.Res_25 := FALSE;
   BB_SHL_G3.Bef.Res_26 := FALSE;
   BB_SHL_G3.Bef.Res_27 := FALSE;
   BB_SHL_G3.Bef.Res_28 := FALSE;
   BB_SHL_G3.Bef.Res_29 := FALSE;
   BB_SHL_G3.Bef.BF_Set_SW_chg := FALSE;
   BB_SHL_G3.Bef.BF_Quit := FALSE;
   BB_SHL_G3.SW_Hand := 0.0;
   BB_AV.Bef.Bed_Res := FALSE;
   BB_AV.Bef.Bed_UV := FALSE;
   BB_AV.Bef.Bed_NHV := FALSE;
   BB_AV.Bef.Bed_PLS := FALSE;
   BB_AV.Bef.BA_Hand := FALSE;
   BB_AV.Bef.BA_Auto := FALSE;
   BB_AV.Bef.BF_Ein1 := FALSE;
   BB_AV.Bef.BF_Ein2 := FALSE;
   BB_AV.Bef.BF_Aus := FALSE;
   BB_AV.Bef.BZ_Res := FALSE;
   BB_AV.Bef.Res_10 := FALSE;
   BB_AV.Bef.Res_11 := FALSE;
   BB_AV.Bef.Res_12 := FALSE;
   BB_AV.Bef.Res_13 := FALSE;
   BB_AV.Bef.Res_14 := FALSE;
   BB_AV.Bef.Res_15 := FALSE;
   BB_AV.Bef.Res_16 := FALSE;
   BB_AV.Bef.Res_17 := FALSE;
   BB_AV.Bef.Res_18 := FALSE;
   BB_AV.Bef.Res_19 := FALSE;
   BB_AV.Bef.Res_20 := FALSE;
   BB_AV.Bef.Res_21 := FALSE;
   BB_AV.Bef.Res_22 := FALSE;
   BB_AV.Bef.Res_23 := FALSE;
   BB_AV.Bef.Res_24 := FALSE;
   BB_AV.Bef.Res_25 := FALSE;
   BB_AV.Bef.Res_26 := FALSE;
   BB_AV.Bef.Res_27 := FALSE;
   BB_AV.Bef.Res_28 := FALSE;
   BB_AV.Bef.Res_29 := FALSE;
   BB_AV.Bef.BF_Set_SW_chg := FALSE;
   BB_AV.Bef.BF_Quit := FALSE;
   BB_AV.SW_Hand := 0.0;
   BB_LS1.Bef.Bed_Res := FALSE;
   BB_LS1.Bef.Bed_UV := FALSE;
   BB_LS1.Bef.Bed_NHV := FALSE;
   BB_LS1.Bef.Bed_PLS := FALSE;
   BB_LS1.Bef.BA_Hand := FALSE;
   BB_LS1.Bef.BA_Auto := FALSE;
   BB_LS1.Bef.BF_Ein1 := FALSE;
   BB_LS1.Bef.BF_Ein2 := FALSE;
   BB_LS1.Bef.BF_Aus := FALSE;
   BB_LS1.Bef.BZ_Res := FALSE;
   BB_LS1.Bef.Res_10 := FALSE;
   BB_LS1.Bef.Res_11 := FALSE;
   BB_LS1.Bef.Res_12 := FALSE;
   BB_LS1.Bef.Res_13 := FALSE;
   BB_LS1.Bef.Res_14 := FALSE;
   BB_LS1.Bef.Res_15 := FALSE;
   BB_LS1.Bef.Res_16 := FALSE;
   BB_LS1.Bef.Res_17 := FALSE;
   BB_LS1.Bef.Res_18 := FALSE;
   BB_LS1.Bef.Res_19 := FALSE;
   BB_LS1.Bef.Res_20 := FALSE;
   BB_LS1.Bef.Res_21 := FALSE;
   BB_LS1.Bef.Res_22 := FALSE;
   BB_LS1.Bef.Res_23 := FALSE;
   BB_LS1.Bef.Res_24 := FALSE;
   BB_LS1.Bef.Res_25 := FALSE;
   BB_LS1.Bef.Res_26 := FALSE;
   BB_LS1.Bef.Res_27 := FALSE;
   BB_LS1.Bef.Res_28 := FALSE;
   BB_LS1.Bef.Res_29 := FALSE;
   BB_LS1.Bef.BF_Set_SW_chg := FALSE;
   BB_LS1.Bef.BF_Quit := FALSE;
   BB_LS1.SW_Hand := 0.0;
   BB_LS2.Bef.Bed_Res := FALSE;
   BB_LS2.Bef.Bed_UV := FALSE;
   BB_LS2.Bef.Bed_NHV := FALSE;
   BB_LS2.Bef.Bed_PLS := FALSE;
   BB_LS2.Bef.BA_Hand := FALSE;
   BB_LS2.Bef.BA_Auto := FALSE;
   BB_LS2.Bef.BF_Ein1 := FALSE;
   BB_LS2.Bef.BF_Ein2 := FALSE;
   BB_LS2.Bef.BF_Aus := FALSE;
   BB_LS2.Bef.BZ_Res := FALSE;
   BB_LS2.Bef.Res_10 := FALSE;
   BB_LS2.Bef.Res_11 := FALSE;
   BB_LS2.Bef.Res_12 := FALSE;
   BB_LS2.Bef.Res_13 := FALSE;
   BB_LS2.Bef.Res_14 := FALSE;
   BB_LS2.Bef.Res_15 := FALSE;
   BB_LS2.Bef.Res_16 := FALSE;
   BB_LS2.Bef.Res_17 := FALSE;
   BB_LS2.Bef.Res_18 := FALSE;
   BB_LS2.Bef.Res_19 := FALSE;
   BB_LS2.Bef.Res_20 := FALSE;
   BB_LS2.Bef.Res_21 := FALSE;
   BB_LS2.Bef.Res_22 := FALSE;
   BB_LS2.Bef.Res_23 := FALSE;
   BB_LS2.Bef.Res_24 := FALSE;
   BB_LS2.Bef.Res_25 := FALSE;
   BB_LS2.Bef.Res_26 := FALSE;
   BB_LS2.Bef.Res_27 := FALSE;
   BB_LS2.Bef.Res_28 := FALSE;
   BB_LS2.Bef.Res_29 := FALSE;
   BB_LS2.Bef.BF_Set_SW_chg := FALSE;
   BB_LS2.Bef.BF_Quit := FALSE;
   BB_LS2.SW_Hand := 0.0;
   BB1_RZP1.Bef.Bed_Res := FALSE;
   BB1_RZP1.Bef.Bed_UV := FALSE;
   BB1_RZP1.Bef.Bed_NHV := FALSE;
   BB1_RZP1.Bef.Bed_PLS := FALSE;
   BB1_RZP1.Bef.BA_Hand := FALSE;
   BB1_RZP1.Bef.BA_Auto := FALSE;
   BB1_RZP1.Bef.BF_Ein1 := FALSE;
   BB1_RZP1.Bef.BF_Ein2 := FALSE;
   BB1_RZP1.Bef.BF_Aus := FALSE;
   BB1_RZP1.Bef.BZ_Res := FALSE;
   BB1_RZP1.Bef.Res_10 := FALSE;
   BB1_RZP1.Bef.Res_11 := FALSE;
   BB1_RZP1.Bef.Res_12 := FALSE;
   BB1_RZP1.Bef.Res_13 := FALSE;
   BB1_RZP1.Bef.Res_14 := FALSE;
   BB1_RZP1.Bef.Res_15 := FALSE;
   BB1_RZP1.Bef.Res_16 := FALSE;
   BB1_RZP1.Bef.Res_17 := FALSE;
   BB1_RZP1.Bef.Res_18 := FALSE;
   BB1_RZP1.Bef.Res_19 := FALSE;
   BB1_RZP1.Bef.Res_20 := FALSE;
   BB1_RZP1.Bef.Res_21 := FALSE;
   BB1_RZP1.Bef.Res_22 := FALSE;
   BB1_RZP1.Bef.Res_23 := FALSE;
   BB1_RZP1.Bef.Res_24 := FALSE;
   BB1_RZP1.Bef.Res_25 := FALSE;
   BB1_RZP1.Bef.Res_26 := FALSE;
   BB1_RZP1.Bef.Res_27 := FALSE;
   BB1_RZP1.Bef.Res_28 := FALSE;
   BB1_RZP1.Bef.Res_29 := FALSE;
   BB1_RZP1.Bef.BF_Set_SW_chg := FALSE;
   BB1_RZP1.Bef.BF_Quit := FALSE;
   BB1_RZP1.SW_Hand := 0.0;
   BB1_RZP2.Bef.Bed_Res := FALSE;
   BB1_RZP2.Bef.Bed_UV := FALSE;
   BB1_RZP2.Bef.Bed_NHV := FALSE;
   BB1_RZP2.Bef.Bed_PLS := FALSE;
   BB1_RZP2.Bef.BA_Hand := FALSE;
   BB1_RZP2.Bef.BA_Auto := FALSE;
   BB1_RZP2.Bef.BF_Ein1 := FALSE;
   BB1_RZP2.Bef.BF_Ein2 := FALSE;
   BB1_RZP2.Bef.BF_Aus := FALSE;
   BB1_RZP2.Bef.BZ_Res := FALSE;
   BB1_RZP2.Bef.Res_10 := FALSE;
   BB1_RZP2.Bef.Res_11 := FALSE;
   BB1_RZP2.Bef.Res_12 := FALSE;
   BB1_RZP2.Bef.Res_13 := FALSE;
   BB1_RZP2.Bef.Res_14 := FALSE;
   BB1_RZP2.Bef.Res_15 := FALSE;
   BB1_RZP2.Bef.Res_16 := FALSE;
   BB1_RZP2.Bef.Res_17 := FALSE;
   BB1_RZP2.Bef.Res_18 := FALSE;
   BB1_RZP2.Bef.Res_19 := FALSE;
   BB1_RZP2.Bef.Res_20 := FALSE;
   BB1_RZP2.Bef.Res_21 := FALSE;
   BB1_RZP2.Bef.Res_22 := FALSE;
   BB1_RZP2.Bef.Res_23 := FALSE;
   BB1_RZP2.Bef.Res_24 := FALSE;
   BB1_RZP2.Bef.Res_25 := FALSE;
   BB1_RZP2.Bef.Res_26 := FALSE;
   BB1_RZP2.Bef.Res_27 := FALSE;
   BB1_RZP2.Bef.Res_28 := FALSE;
   BB1_RZP2.Bef.Res_29 := FALSE;
   BB1_RZP2.Bef.BF_Set_SW_chg := FALSE;
   BB1_RZP2.Bef.BF_Quit := FALSE;
   BB1_RZP2.SW_Hand := 0.0;
   BB1_UeSP.Bef.Bed_Res := FALSE;
   BB1_UeSP.Bef.Bed_UV := FALSE;
   BB1_UeSP.Bef.Bed_NHV := FALSE;
   BB1_UeSP.Bef.Bed_PLS := FALSE;
   BB1_UeSP.Bef.BA_Hand := FALSE;
   BB1_UeSP.Bef.BA_Auto := FALSE;
   BB1_UeSP.Bef.BF_Ein1 := FALSE;
   BB1_UeSP.Bef.BF_Ein2 := FALSE;
   BB1_UeSP.Bef.BF_Aus := FALSE;
   BB1_UeSP.Bef.BZ_Res := FALSE;
   BB1_UeSP.Bef.Res_10 := FALSE;
   BB1_UeSP.Bef.Res_11 := FALSE;
   BB1_UeSP.Bef.Res_12 := FALSE;
   BB1_UeSP.Bef.Res_13 := FALSE;
   BB1_UeSP.Bef.Res_14 := FALSE;
   BB1_UeSP.Bef.Res_15 := FALSE;
   BB1_UeSP.Bef.Res_16 := FALSE;
   BB1_UeSP.Bef.Res_17 := FALSE;
   BB1_UeSP.Bef.Res_18 := FALSE;
   BB1_UeSP.Bef.Res_19 := FALSE;
   BB1_UeSP.Bef.Res_20 := FALSE;
   BB1_UeSP.Bef.Res_21 := FALSE;
   BB1_UeSP.Bef.Res_22 := FALSE;
   BB1_UeSP.Bef.Res_23 := FALSE;
   BB1_UeSP.Bef.Res_24 := FALSE;
   BB1_UeSP.Bef.Res_25 := FALSE;
   BB1_UeSP.Bef.Res_26 := FALSE;
   BB1_UeSP.Bef.Res_27 := FALSE;
   BB1_UeSP.Bef.Res_28 := FALSE;
   BB1_UeSP.Bef.Res_29 := FALSE;
   BB1_UeSP.Bef.BF_Set_SW_chg := FALSE;
   BB1_UeSP.Bef.BF_Quit := FALSE;
   BB1_UeSP.SW_Hand := 0.0;
   BB1_AS1.Bef.Bed_Res := FALSE;
   BB1_AS1.Bef.Bed_UV := FALSE;
   BB1_AS1.Bef.Bed_NHV := FALSE;
   BB1_AS1.Bef.Bed_PLS := FALSE;
   BB1_AS1.Bef.BA_Hand := FALSE;
   BB1_AS1.Bef.BA_Auto := FALSE;
   BB1_AS1.Bef.BF_Ein1 := FALSE;
   BB1_AS1.Bef.BF_Ein2 := FALSE;
   BB1_AS1.Bef.BF_Aus := FALSE;
   BB1_AS1.Bef.BZ_Res := FALSE;
   BB1_AS1.Bef.Res_10 := FALSE;
   BB1_AS1.Bef.Res_11 := FALSE;
   BB1_AS1.Bef.Res_12 := FALSE;
   BB1_AS1.Bef.Res_13 := FALSE;
   BB1_AS1.Bef.Res_14 := FALSE;
   BB1_AS1.Bef.Res_15 := FALSE;
   BB1_AS1.Bef.Res_16 := FALSE;
   BB1_AS1.Bef.Res_17 := FALSE;
   BB1_AS1.Bef.Res_18 := FALSE;
   BB1_AS1.Bef.Res_19 := FALSE;
   BB1_AS1.Bef.Res_20 := FALSE;
   BB1_AS1.Bef.Res_21 := FALSE;
   BB1_AS1.Bef.Res_22 := FALSE;
   BB1_AS1.Bef.Res_23 := FALSE;
   BB1_AS1.Bef.Res_24 := FALSE;
   BB1_AS1.Bef.Res_25 := FALSE;
   BB1_AS1.Bef.Res_26 := FALSE;
   BB1_AS1.Bef.Res_27 := FALSE;
   BB1_AS1.Bef.Res_28 := FALSE;
   BB1_AS1.Bef.Res_29 := FALSE;
   BB1_AS1.Bef.BF_Set_SW_chg := FALSE;
   BB1_AS1.Bef.BF_Quit := FALSE;
   BB1_AS1.SW_Hand := 0.0;
   BB1_AS2.Bef.Bed_Res := FALSE;
   BB1_AS2.Bef.Bed_UV := FALSE;
   BB1_AS2.Bef.Bed_NHV := FALSE;
   BB1_AS2.Bef.Bed_PLS := FALSE;
   BB1_AS2.Bef.BA_Hand := FALSE;
   BB1_AS2.Bef.BA_Auto := FALSE;
   BB1_AS2.Bef.BF_Ein1 := FALSE;
   BB1_AS2.Bef.BF_Ein2 := FALSE;
   BB1_AS2.Bef.BF_Aus := FALSE;
   BB1_AS2.Bef.BZ_Res := FALSE;
   BB1_AS2.Bef.Res_10 := FALSE;
   BB1_AS2.Bef.Res_11 := FALSE;
   BB1_AS2.Bef.Res_12 := FALSE;
   BB1_AS2.Bef.Res_13 := FALSE;
   BB1_AS2.Bef.Res_14 := FALSE;
   BB1_AS2.Bef.Res_15 := FALSE;
   BB1_AS2.Bef.Res_16 := FALSE;
   BB1_AS2.Bef.Res_17 := FALSE;
   BB1_AS2.Bef.Res_18 := FALSE;
   BB1_AS2.Bef.Res_19 := FALSE;
   BB1_AS2.Bef.Res_20 := FALSE;
   BB1_AS2.Bef.Res_21 := FALSE;
   BB1_AS2.Bef.Res_22 := FALSE;
   BB1_AS2.Bef.Res_23 := FALSE;
   BB1_AS2.Bef.Res_24 := FALSE;
   BB1_AS2.Bef.Res_25 := FALSE;
   BB1_AS2.Bef.Res_26 := FALSE;
   BB1_AS2.Bef.Res_27 := FALSE;
   BB1_AS2.Bef.Res_28 := FALSE;
   BB1_AS2.Bef.Res_29 := FALSE;
   BB1_AS2.Bef.BF_Set_SW_chg := FALSE;
   BB1_AS2.Bef.BF_Quit := FALSE;
   BB1_AS2.SW_Hand := 0.0;
   BB1_SR1.Bef.Bed_Res := FALSE;
   BB1_SR1.Bef.Bed_UV := FALSE;
   BB1_SR1.Bef.Bed_NHV := FALSE;
   BB1_SR1.Bef.Bed_PLS := FALSE;
   BB1_SR1.Bef.BA_Hand := FALSE;
   BB1_SR1.Bef.BA_Auto := FALSE;
   BB1_SR1.Bef.BF_Ein1 := FALSE;
   BB1_SR1.Bef.BF_Ein2 := FALSE;
   BB1_SR1.Bef.BF_Aus := FALSE;
   BB1_SR1.Bef.BZ_Res := FALSE;
   BB1_SR1.Bef.Res_10 := FALSE;
   BB1_SR1.Bef.Res_11 := FALSE;
   BB1_SR1.Bef.Res_12 := FALSE;
   BB1_SR1.Bef.Res_13 := FALSE;
   BB1_SR1.Bef.Res_14 := FALSE;
   BB1_SR1.Bef.Res_15 := FALSE;
   BB1_SR1.Bef.Res_16 := FALSE;
   BB1_SR1.Bef.Res_17 := FALSE;
   BB1_SR1.Bef.Res_18 := FALSE;
   BB1_SR1.Bef.Res_19 := FALSE;
   BB1_SR1.Bef.Res_20 := FALSE;
   BB1_SR1.Bef.Res_21 := FALSE;
   BB1_SR1.Bef.Res_22 := FALSE;
   BB1_SR1.Bef.Res_23 := FALSE;
   BB1_SR1.Bef.Res_24 := FALSE;
   BB1_SR1.Bef.Res_25 := FALSE;
   BB1_SR1.Bef.Res_26 := FALSE;
   BB1_SR1.Bef.Res_27 := FALSE;
   BB1_SR1.Bef.Res_28 := FALSE;
   BB1_SR1.Bef.Res_29 := FALSE;
   BB1_SR1.Bef.BF_Set_SW_chg := FALSE;
   BB1_SR1.Bef.BF_Quit := FALSE;
   BB1_SR1.SW_Hand := 0.0;
   BB1_SR2.Bef.Bed_Res := FALSE;
   BB1_SR2.Bef.Bed_UV := FALSE;
   BB1_SR2.Bef.Bed_NHV := FALSE;
   BB1_SR2.Bef.Bed_PLS := FALSE;
   BB1_SR2.Bef.BA_Hand := FALSE;
   BB1_SR2.Bef.BA_Auto := FALSE;
   BB1_SR2.Bef.BF_Ein1 := FALSE;
   BB1_SR2.Bef.BF_Ein2 := FALSE;
   BB1_SR2.Bef.BF_Aus := FALSE;
   BB1_SR2.Bef.BZ_Res := FALSE;
   BB1_SR2.Bef.Res_10 := FALSE;
   BB1_SR2.Bef.Res_11 := FALSE;
   BB1_SR2.Bef.Res_12 := FALSE;
   BB1_SR2.Bef.Res_13 := FALSE;
   BB1_SR2.Bef.Res_14 := FALSE;
   BB1_SR2.Bef.Res_15 := FALSE;
   BB1_SR2.Bef.Res_16 := FALSE;
   BB1_SR2.Bef.Res_17 := FALSE;
   BB1_SR2.Bef.Res_18 := FALSE;
   BB1_SR2.Bef.Res_19 := FALSE;
   BB1_SR2.Bef.Res_20 := FALSE;
   BB1_SR2.Bef.Res_21 := FALSE;
   BB1_SR2.Bef.Res_22 := FALSE;
   BB1_SR2.Bef.Res_23 := FALSE;
   BB1_SR2.Bef.Res_24 := FALSE;
   BB1_SR2.Bef.Res_25 := FALSE;
   BB1_SR2.Bef.Res_26 := FALSE;
   BB1_SR2.Bef.Res_27 := FALSE;
   BB1_SR2.Bef.Res_28 := FALSE;
   BB1_SR2.Bef.Res_29 := FALSE;
   BB1_SR2.Bef.BF_Set_SW_chg := FALSE;
   BB1_SR2.Bef.BF_Quit := FALSE;
   BB1_SR2.SW_Hand := 0.0;
   BB2_RZP1.Bef.Bed_Res := FALSE;
   BB2_RZP1.Bef.Bed_UV := FALSE;
   BB2_RZP1.Bef.Bed_NHV := FALSE;
   BB2_RZP1.Bef.Bed_PLS := FALSE;
   BB2_RZP1.Bef.BA_Hand := FALSE;
   BB2_RZP1.Bef.BA_Auto := FALSE;
   BB2_RZP1.Bef.BF_Ein1 := FALSE;
   BB2_RZP1.Bef.BF_Ein2 := FALSE;
   BB2_RZP1.Bef.BF_Aus := FALSE;
   BB2_RZP1.Bef.BZ_Res := FALSE;
   BB2_RZP1.Bef.Res_10 := FALSE;
   BB2_RZP1.Bef.Res_11 := FALSE;
   BB2_RZP1.Bef.Res_12 := FALSE;
   BB2_RZP1.Bef.Res_13 := FALSE;
   BB2_RZP1.Bef.Res_14 := FALSE;
   BB2_RZP1.Bef.Res_15 := FALSE;
   BB2_RZP1.Bef.Res_16 := FALSE;
   BB2_RZP1.Bef.Res_17 := FALSE;
   BB2_RZP1.Bef.Res_18 := FALSE;
   BB2_RZP1.Bef.Res_19 := FALSE;
   BB2_RZP1.Bef.Res_20 := FALSE;
   BB2_RZP1.Bef.Res_21 := FALSE;
   BB2_RZP1.Bef.Res_22 := FALSE;
   BB2_RZP1.Bef.Res_23 := FALSE;
   BB2_RZP1.Bef.Res_24 := FALSE;
   BB2_RZP1.Bef.Res_25 := FALSE;
   BB2_RZP1.Bef.Res_26 := FALSE;
   BB2_RZP1.Bef.Res_27 := FALSE;
   BB2_RZP1.Bef.Res_28 := FALSE;
   BB2_RZP1.Bef.Res_29 := FALSE;
   BB2_RZP1.Bef.BF_Set_SW_chg := FALSE;
   BB2_RZP1.Bef.BF_Quit := FALSE;
   BB2_RZP1.SW_Hand := 0.0;
   BB2_RZP2.Bef.Bed_Res := FALSE;
   BB2_RZP2.Bef.Bed_UV := FALSE;
   BB2_RZP2.Bef.Bed_NHV := FALSE;
   BB2_RZP2.Bef.Bed_PLS := FALSE;
   BB2_RZP2.Bef.BA_Hand := FALSE;
   BB2_RZP2.Bef.BA_Auto := FALSE;
   BB2_RZP2.Bef.BF_Ein1 := FALSE;
   BB2_RZP2.Bef.BF_Ein2 := FALSE;
   BB2_RZP2.Bef.BF_Aus := FALSE;
   BB2_RZP2.Bef.BZ_Res := FALSE;
   BB2_RZP2.Bef.Res_10 := FALSE;
   BB2_RZP2.Bef.Res_11 := FALSE;
   BB2_RZP2.Bef.Res_12 := FALSE;
   BB2_RZP2.Bef.Res_13 := FALSE;
   BB2_RZP2.Bef.Res_14 := FALSE;
   BB2_RZP2.Bef.Res_15 := FALSE;
   BB2_RZP2.Bef.Res_16 := FALSE;
   BB2_RZP2.Bef.Res_17 := FALSE;
   BB2_RZP2.Bef.Res_18 := FALSE;
   BB2_RZP2.Bef.Res_19 := FALSE;
   BB2_RZP2.Bef.Res_20 := FALSE;
   BB2_RZP2.Bef.Res_21 := FALSE;
   BB2_RZP2.Bef.Res_22 := FALSE;
   BB2_RZP2.Bef.Res_23 := FALSE;
   BB2_RZP2.Bef.Res_24 := FALSE;
   BB2_RZP2.Bef.Res_25 := FALSE;
   BB2_RZP2.Bef.Res_26 := FALSE;
   BB2_RZP2.Bef.Res_27 := FALSE;
   BB2_RZP2.Bef.Res_28 := FALSE;
   BB2_RZP2.Bef.Res_29 := FALSE;
   BB2_RZP2.Bef.BF_Set_SW_chg := FALSE;
   BB2_RZP2.Bef.BF_Quit := FALSE;
   BB2_RZP2.SW_Hand := 0.0;
   BB2_UeSP.Bef.Bed_Res := FALSE;
   BB2_UeSP.Bef.Bed_UV := FALSE;
   BB2_UeSP.Bef.Bed_NHV := FALSE;
   BB2_UeSP.Bef.Bed_PLS := FALSE;
   BB2_UeSP.Bef.BA_Hand := FALSE;
   BB2_UeSP.Bef.BA_Auto := FALSE;
   BB2_UeSP.Bef.BF_Ein1 := FALSE;
   BB2_UeSP.Bef.BF_Ein2 := FALSE;
   BB2_UeSP.Bef.BF_Aus := FALSE;
   BB2_UeSP.Bef.BZ_Res := FALSE;
   BB2_UeSP.Bef.Res_10 := FALSE;
   BB2_UeSP.Bef.Res_11 := FALSE;
   BB2_UeSP.Bef.Res_12 := FALSE;
   BB2_UeSP.Bef.Res_13 := FALSE;
   BB2_UeSP.Bef.Res_14 := FALSE;
   BB2_UeSP.Bef.Res_15 := FALSE;
   BB2_UeSP.Bef.Res_16 := FALSE;
   BB2_UeSP.Bef.Res_17 := FALSE;
   BB2_UeSP.Bef.Res_18 := FALSE;
   BB2_UeSP.Bef.Res_19 := FALSE;
   BB2_UeSP.Bef.Res_20 := FALSE;
   BB2_UeSP.Bef.Res_21 := FALSE;
   BB2_UeSP.Bef.Res_22 := FALSE;
   BB2_UeSP.Bef.Res_23 := FALSE;
   BB2_UeSP.Bef.Res_24 := FALSE;
   BB2_UeSP.Bef.Res_25 := FALSE;
   BB2_UeSP.Bef.Res_26 := FALSE;
   BB2_UeSP.Bef.Res_27 := FALSE;
   BB2_UeSP.Bef.Res_28 := FALSE;
   BB2_UeSP.Bef.Res_29 := FALSE;
   BB2_UeSP.Bef.BF_Set_SW_chg := FALSE;
   BB2_UeSP.Bef.BF_Quit := FALSE;
   BB2_UeSP.SW_Hand := 0.0;
   BB2_AS1.Bef.Bed_Res := FALSE;
   BB2_AS1.Bef.Bed_UV := FALSE;
   BB2_AS1.Bef.Bed_NHV := FALSE;
   BB2_AS1.Bef.Bed_PLS := FALSE;
   BB2_AS1.Bef.BA_Hand := FALSE;
   BB2_AS1.Bef.BA_Auto := FALSE;
   BB2_AS1.Bef.BF_Ein1 := FALSE;
   BB2_AS1.Bef.BF_Ein2 := FALSE;
   BB2_AS1.Bef.BF_Aus := FALSE;
   BB2_AS1.Bef.BZ_Res := FALSE;
   BB2_AS1.Bef.Res_10 := FALSE;
   BB2_AS1.Bef.Res_11 := FALSE;
   BB2_AS1.Bef.Res_12 := FALSE;
   BB2_AS1.Bef.Res_13 := FALSE;
   BB2_AS1.Bef.Res_14 := FALSE;
   BB2_AS1.Bef.Res_15 := FALSE;
   BB2_AS1.Bef.Res_16 := FALSE;
   BB2_AS1.Bef.Res_17 := FALSE;
   BB2_AS1.Bef.Res_18 := FALSE;
   BB2_AS1.Bef.Res_19 := FALSE;
   BB2_AS1.Bef.Res_20 := FALSE;
   BB2_AS1.Bef.Res_21 := FALSE;
   BB2_AS1.Bef.Res_22 := FALSE;
   BB2_AS1.Bef.Res_23 := FALSE;
   BB2_AS1.Bef.Res_24 := FALSE;
   BB2_AS1.Bef.Res_25 := FALSE;
   BB2_AS1.Bef.Res_26 := FALSE;
   BB2_AS1.Bef.Res_27 := FALSE;
   BB2_AS1.Bef.Res_28 := FALSE;
   BB2_AS1.Bef.Res_29 := FALSE;
   BB2_AS1.Bef.BF_Set_SW_chg := FALSE;
   BB2_AS1.Bef.BF_Quit := FALSE;
   BB2_AS1.SW_Hand := 0.0;
   BB2_AS2.Bef.Bed_Res := FALSE;
   BB2_AS2.Bef.Bed_UV := FALSE;
   BB2_AS2.Bef.Bed_NHV := FALSE;
   BB2_AS2.Bef.Bed_PLS := FALSE;
   BB2_AS2.Bef.BA_Hand := FALSE;
   BB2_AS2.Bef.BA_Auto := FALSE;
   BB2_AS2.Bef.BF_Ein1 := FALSE;
   BB2_AS2.Bef.BF_Ein2 := FALSE;
   BB2_AS2.Bef.BF_Aus := FALSE;
   BB2_AS2.Bef.BZ_Res := FALSE;
   BB2_AS2.Bef.Res_10 := FALSE;
   BB2_AS2.Bef.Res_11 := FALSE;
   BB2_AS2.Bef.Res_12 := FALSE;
   BB2_AS2.Bef.Res_13 := FALSE;
   BB2_AS2.Bef.Res_14 := FALSE;
   BB2_AS2.Bef.Res_15 := FALSE;
   BB2_AS2.Bef.Res_16 := FALSE;
   BB2_AS2.Bef.Res_17 := FALSE;
   BB2_AS2.Bef.Res_18 := FALSE;
   BB2_AS2.Bef.Res_19 := FALSE;
   BB2_AS2.Bef.Res_20 := FALSE;
   BB2_AS2.Bef.Res_21 := FALSE;
   BB2_AS2.Bef.Res_22 := FALSE;
   BB2_AS2.Bef.Res_23 := FALSE;
   BB2_AS2.Bef.Res_24 := FALSE;
   BB2_AS2.Bef.Res_25 := FALSE;
   BB2_AS2.Bef.Res_26 := FALSE;
   BB2_AS2.Bef.Res_27 := FALSE;
   BB2_AS2.Bef.Res_28 := FALSE;
   BB2_AS2.Bef.Res_29 := FALSE;
   BB2_AS2.Bef.BF_Set_SW_chg := FALSE;
   BB2_AS2.Bef.BF_Quit := FALSE;
   BB2_AS2.SW_Hand := 0.0;
   BB2_SR1.Bef.Bed_Res := FALSE;
   BB2_SR1.Bef.Bed_UV := FALSE;
   BB2_SR1.Bef.Bed_NHV := FALSE;
   BB2_SR1.Bef.Bed_PLS := FALSE;
   BB2_SR1.Bef.BA_Hand := FALSE;
   BB2_SR1.Bef.BA_Auto := FALSE;
   BB2_SR1.Bef.BF_Ein1 := FALSE;
   BB2_SR1.Bef.BF_Ein2 := FALSE;
   BB2_SR1.Bef.BF_Aus := FALSE;
   BB2_SR1.Bef.BZ_Res := FALSE;
   BB2_SR1.Bef.Res_10 := FALSE;
   BB2_SR1.Bef.Res_11 := FALSE;
   BB2_SR1.Bef.Res_12 := FALSE;
   BB2_SR1.Bef.Res_13 := FALSE;
   BB2_SR1.Bef.Res_14 := FALSE;
   BB2_SR1.Bef.Res_15 := FALSE;
   BB2_SR1.Bef.Res_16 := FALSE;
   BB2_SR1.Bef.Res_17 := FALSE;
   BB2_SR1.Bef.Res_18 := FALSE;
   BB2_SR1.Bef.Res_19 := FALSE;
   BB2_SR1.Bef.Res_20 := FALSE;
   BB2_SR1.Bef.Res_21 := FALSE;
   BB2_SR1.Bef.Res_22 := FALSE;
   BB2_SR1.Bef.Res_23 := FALSE;
   BB2_SR1.Bef.Res_24 := FALSE;
   BB2_SR1.Bef.Res_25 := FALSE;
   BB2_SR1.Bef.Res_26 := FALSE;
   BB2_SR1.Bef.Res_27 := FALSE;
   BB2_SR1.Bef.Res_28 := FALSE;
   BB2_SR1.Bef.Res_29 := FALSE;
   BB2_SR1.Bef.BF_Set_SW_chg := FALSE;
   BB2_SR1.Bef.BF_Quit := FALSE;
   BB2_SR1.SW_Hand := 0.0;
   BB2_SR2.Bef.Bed_Res := FALSE;
   BB2_SR2.Bef.Bed_UV := FALSE;
   BB2_SR2.Bef.Bed_NHV := FALSE;
   BB2_SR2.Bef.Bed_PLS := FALSE;
   BB2_SR2.Bef.BA_Hand := FALSE;
   BB2_SR2.Bef.BA_Auto := FALSE;
   BB2_SR2.Bef.BF_Ein1 := FALSE;
   BB2_SR2.Bef.BF_Ein2 := FALSE;
   BB2_SR2.Bef.BF_Aus := FALSE;
   BB2_SR2.Bef.BZ_Res := FALSE;
   BB2_SR2.Bef.Res_10 := FALSE;
   BB2_SR2.Bef.Res_11 := FALSE;
   BB2_SR2.Bef.Res_12 := FALSE;
   BB2_SR2.Bef.Res_13 := FALSE;
   BB2_SR2.Bef.Res_14 := FALSE;
   BB2_SR2.Bef.Res_15 := FALSE;
   BB2_SR2.Bef.Res_16 := FALSE;
   BB2_SR2.Bef.Res_17 := FALSE;
   BB2_SR2.Bef.Res_18 := FALSE;
   BB2_SR2.Bef.Res_19 := FALSE;
   BB2_SR2.Bef.Res_20 := FALSE;
   BB2_SR2.Bef.Res_21 := FALSE;
   BB2_SR2.Bef.Res_22 := FALSE;
   BB2_SR2.Bef.Res_23 := FALSE;
   BB2_SR2.Bef.Res_24 := FALSE;
   BB2_SR2.Bef.Res_25 := FALSE;
   BB2_SR2.Bef.Res_26 := FALSE;
   BB2_SR2.Bef.Res_27 := FALSE;
   BB2_SR2.Bef.Res_28 := FALSE;
   BB2_SR2.Bef.Res_29 := FALSE;
   BB2_SR2.Bef.BF_Set_SW_chg := FALSE;
   BB2_SR2.Bef.BF_Quit := FALSE;
   BB2_SR2.SW_Hand := 0.0;
   BB1_SR_K.Bef.Bed_Res := FALSE;
   BB1_SR_K.Bef.Bed_UV := FALSE;
   BB1_SR_K.Bef.Bed_NHV := FALSE;
   BB1_SR_K.Bef.Bed_PLS := FALSE;
   BB1_SR_K.Bef.BA_Hand := FALSE;
   BB1_SR_K.Bef.BA_Auto := FALSE;
   BB1_SR_K.Bef.BF_Ein1 := FALSE;
   BB1_SR_K.Bef.BF_Ein2 := FALSE;
   BB1_SR_K.Bef.BF_Aus := FALSE;
   BB1_SR_K.Bef.BZ_Res := FALSE;
   BB1_SR_K.Bef.Res_10 := FALSE;
   BB1_SR_K.Bef.Res_11 := FALSE;
   BB1_SR_K.Bef.Res_12 := FALSE;
   BB1_SR_K.Bef.Res_13 := FALSE;
   BB1_SR_K.Bef.Res_14 := FALSE;
   BB1_SR_K.Bef.Res_15 := FALSE;
   BB1_SR_K.Bef.Res_16 := FALSE;
   BB1_SR_K.Bef.Res_17 := FALSE;
   BB1_SR_K.Bef.Res_18 := FALSE;
   BB1_SR_K.Bef.Res_19 := FALSE;
   BB1_SR_K.Bef.Res_20 := FALSE;
   BB1_SR_K.Bef.Res_21 := FALSE;
   BB1_SR_K.Bef.Res_22 := FALSE;
   BB1_SR_K.Bef.Res_23 := FALSE;
   BB1_SR_K.Bef.Res_24 := FALSE;
   BB1_SR_K.Bef.Res_25 := FALSE;
   BB1_SR_K.Bef.Res_26 := FALSE;
   BB1_SR_K.Bef.Res_27 := FALSE;
   BB1_SR_K.Bef.Res_28 := FALSE;
   BB1_SR_K.Bef.Res_29 := FALSE;
   BB1_SR_K.Bef.BF_Set_SW_chg := FALSE;
   BB1_SR_K.Bef.BF_Quit := FALSE;
   BB1_SR_K.SW_Hand := 0.0;
   Zulauf_AR_P1.Bef.Bed_Res := FALSE;
   Zulauf_AR_P1.Bef.Bed_UV := FALSE;
   Zulauf_AR_P1.Bef.Bed_NHV := FALSE;
   Zulauf_AR_P1.Bef.Bed_PLS := FALSE;
   Zulauf_AR_P1.Bef.BA_Hand := FALSE;
   Zulauf_AR_P1.Bef.BA_Auto := FALSE;
   Zulauf_AR_P1.Bef.BF_Ein1 := FALSE;
   Zulauf_AR_P1.Bef.BF_Ein2 := FALSE;
   Zulauf_AR_P1.Bef.BF_Aus := FALSE;
   Zulauf_AR_P1.Bef.BZ_Res := FALSE;
   Zulauf_AR_P1.Bef.Res_10 := FALSE;
   Zulauf_AR_P1.Bef.Res_11 := FALSE;
   Zulauf_AR_P1.Bef.Res_12 := FALSE;
   Zulauf_AR_P1.Bef.Res_13 := FALSE;
   Zulauf_AR_P1.Bef.Res_14 := FALSE;
   Zulauf_AR_P1.Bef.Res_15 := FALSE;
   Zulauf_AR_P1.Bef.Res_16 := FALSE;
   Zulauf_AR_P1.Bef.Res_17 := FALSE;
   Zulauf_AR_P1.Bef.Res_18 := FALSE;
   Zulauf_AR_P1.Bef.Res_19 := FALSE;
   Zulauf_AR_P1.Bef.Res_20 := FALSE;
   Zulauf_AR_P1.Bef.Res_21 := FALSE;
   Zulauf_AR_P1.Bef.Res_22 := FALSE;
   Zulauf_AR_P1.Bef.Res_23 := FALSE;
   Zulauf_AR_P1.Bef.Res_24 := FALSE;
   Zulauf_AR_P1.Bef.Res_25 := FALSE;
   Zulauf_AR_P1.Bef.Res_26 := FALSE;
   Zulauf_AR_P1.Bef.Res_27 := FALSE;
   Zulauf_AR_P1.Bef.Res_28 := FALSE;
   Zulauf_AR_P1.Bef.Res_29 := FALSE;
   Zulauf_AR_P1.Bef.BF_Set_SW_chg := FALSE;
   Zulauf_AR_P1.Bef.BF_Quit := FALSE;
   Zulauf_AR_P1.SW_Hand := 0.0;
   Zulauf_AR_P2.Bef.Bed_Res := FALSE;
   Zulauf_AR_P2.Bef.Bed_UV := FALSE;
   Zulauf_AR_P2.Bef.Bed_NHV := FALSE;
   Zulauf_AR_P2.Bef.Bed_PLS := FALSE;
   Zulauf_AR_P2.Bef.BA_Hand := FALSE;
   Zulauf_AR_P2.Bef.BA_Auto := FALSE;
   Zulauf_AR_P2.Bef.BF_Ein1 := FALSE;
   Zulauf_AR_P2.Bef.BF_Ein2 := FALSE;
   Zulauf_AR_P2.Bef.BF_Aus := FALSE;
   Zulauf_AR_P2.Bef.BZ_Res := FALSE;
   Zulauf_AR_P2.Bef.Res_10 := FALSE;
   Zulauf_AR_P2.Bef.Res_11 := FALSE;
   Zulauf_AR_P2.Bef.Res_12 := FALSE;
   Zulauf_AR_P2.Bef.Res_13 := FALSE;
   Zulauf_AR_P2.Bef.Res_14 := FALSE;
   Zulauf_AR_P2.Bef.Res_15 := FALSE;
   Zulauf_AR_P2.Bef.Res_16 := FALSE;
   Zulauf_AR_P2.Bef.Res_17 := FALSE;
   Zulauf_AR_P2.Bef.Res_18 := FALSE;
   Zulauf_AR_P2.Bef.Res_19 := FALSE;
   Zulauf_AR_P2.Bef.Res_20 := FALSE;
   Zulauf_AR_P2.Bef.Res_21 := FALSE;
   Zulauf_AR_P2.Bef.Res_22 := FALSE;
   Zulauf_AR_P2.Bef.Res_23 := FALSE;
   Zulauf_AR_P2.Bef.Res_24 := FALSE;
   Zulauf_AR_P2.Bef.Res_25 := FALSE;
   Zulauf_AR_P2.Bef.Res_26 := FALSE;
   Zulauf_AR_P2.Bef.Res_27 := FALSE;
   Zulauf_AR_P2.Bef.Res_28 := FALSE;
   Zulauf_AR_P2.Bef.Res_29 := FALSE;
   Zulauf_AR_P2.Bef.BF_Set_SW_chg := FALSE;
   Zulauf_AR_P2.Bef.BF_Quit := FALSE;
   Zulauf_AR_P2.SW_Hand := 0.0;
   Zulauf_AS.Bef.Bed_Res := FALSE;
   Zulauf_AS.Bef.Bed_UV := FALSE;
   Zulauf_AS.Bef.Bed_NHV := FALSE;
   Zulauf_AS.Bef.Bed_PLS := FALSE;
   Zulauf_AS.Bef.BA_Hand := FALSE;
   Zulauf_AS.Bef.BA_Auto := FALSE;
   Zulauf_AS.Bef.BF_Ein1 := FALSE;
   Zulauf_AS.Bef.BF_Ein2 := FALSE;
   Zulauf_AS.Bef.BF_Aus := FALSE;
   Zulauf_AS.Bef.BZ_Res := FALSE;
   Zulauf_AS.Bef.Res_10 := FALSE;
   Zulauf_AS.Bef.Res_11 := FALSE;
   Zulauf_AS.Bef.Res_12 := FALSE;
   Zulauf_AS.Bef.Res_13 := FALSE;
   Zulauf_AS.Bef.Res_14 := FALSE;
   Zulauf_AS.Bef.Res_15 := FALSE;
   Zulauf_AS.Bef.Res_16 := FALSE;
   Zulauf_AS.Bef.Res_17 := FALSE;
   Zulauf_AS.Bef.Res_18 := FALSE;
   Zulauf_AS.Bef.Res_19 := FALSE;
   Zulauf_AS.Bef.Res_20 := FALSE;
   Zulauf_AS.Bef.Res_21 := FALSE;
   Zulauf_AS.Bef.Res_22 := FALSE;
   Zulauf_AS.Bef.Res_23 := FALSE;
   Zulauf_AS.Bef.Res_24 := FALSE;
   Zulauf_AS.Bef.Res_25 := FALSE;
   Zulauf_AS.Bef.Res_26 := FALSE;
   Zulauf_AS.Bef.Res_27 := FALSE;
   Zulauf_AS.Bef.Res_28 := FALSE;
   Zulauf_AS.Bef.Res_29 := FALSE;
   Zulauf_AS.Bef.BF_Set_SW_chg := FALSE;
   Zulauf_AS.Bef.BF_Quit := FALSE;
   Zulauf_AS.SW_Hand := 0.0;
   Zulauf_RA_SA.Bef.Bed_Res := FALSE;
   Zulauf_RA_SA.Bef.Bed_UV := FALSE;
   Zulauf_RA_SA.Bef.Bed_NHV := FALSE;
   Zulauf_RA_SA.Bef.Bed_PLS := FALSE;
   Zulauf_RA_SA.Bef.BA_Hand := FALSE;
   Zulauf_RA_SA.Bef.BA_Auto := FALSE;
   Zulauf_RA_SA.Bef.BF_Ein1 := FALSE;
   Zulauf_RA_SA.Bef.BF_Ein2 := FALSE;
   Zulauf_RA_SA.Bef.BF_Aus := FALSE;
   Zulauf_RA_SA.Bef.BZ_Res := FALSE;
   Zulauf_RA_SA.Bef.Res_10 := FALSE;
   Zulauf_RA_SA.Bef.Res_11 := FALSE;
   Zulauf_RA_SA.Bef.Res_12 := FALSE;
   Zulauf_RA_SA.Bef.Res_13 := FALSE;
   Zulauf_RA_SA.Bef.Res_14 := FALSE;
   Zulauf_RA_SA.Bef.Res_15 := FALSE;
   Zulauf_RA_SA.Bef.Res_16 := FALSE;
   Zulauf_RA_SA.Bef.Res_17 := FALSE;
   Zulauf_RA_SA.Bef.Res_18 := FALSE;
   Zulauf_RA_SA.Bef.Res_19 := FALSE;
   Zulauf_RA_SA.Bef.Res_20 := FALSE;
   Zulauf_RA_SA.Bef.Res_21 := FALSE;
   Zulauf_RA_SA.Bef.Res_22 := FALSE;
   Zulauf_RA_SA.Bef.Res_23 := FALSE;
   Zulauf_RA_SA.Bef.Res_24 := FALSE;
   Zulauf_RA_SA.Bef.Res_25 := FALSE;
   Zulauf_RA_SA.Bef.Res_26 := FALSE;
   Zulauf_RA_SA.Bef.Res_27 := FALSE;
   Zulauf_RA_SA.Bef.Res_28 := FALSE;
   Zulauf_RA_SA.Bef.Res_29 := FALSE;
   Zulauf_RA_SA.Bef.BF_Set_SW_chg := FALSE;
   Zulauf_RA_SA.Bef.BF_Quit := FALSE;
   Zulauf_RA_SA.SW_Hand := 0.0;
   Zulauf_RA_HZS.Bef.Bed_Res := FALSE;
   Zulauf_RA_HZS.Bef.Bed_UV := FALSE;
   Zulauf_RA_HZS.Bef.Bed_NHV := FALSE;
   Zulauf_RA_HZS.Bef.Bed_PLS := FALSE;
   Zulauf_RA_HZS.Bef.BA_Hand := FALSE;
   Zulauf_RA_HZS.Bef.BA_Auto := FALSE;
   Zulauf_RA_HZS.Bef.BF_Ein1 := FALSE;
   Zulauf_RA_HZS.Bef.BF_Ein2 := FALSE;
   Zulauf_RA_HZS.Bef.BF_Aus := FALSE;
   Zulauf_RA_HZS.Bef.BZ_Res := FALSE;
   Zulauf_RA_HZS.Bef.Res_10 := FALSE;
   Zulauf_RA_HZS.Bef.Res_11 := FALSE;
   Zulauf_RA_HZS.Bef.Res_12 := FALSE;
   Zulauf_RA_HZS.Bef.Res_13 := FALSE;
   Zulauf_RA_HZS.Bef.Res_14 := FALSE;
   Zulauf_RA_HZS.Bef.Res_15 := FALSE;
   Zulauf_RA_HZS.Bef.Res_16 := FALSE;
   Zulauf_RA_HZS.Bef.Res_17 := FALSE;
   Zulauf_RA_HZS.Bef.Res_18 := FALSE;
   Zulauf_RA_HZS.Bef.Res_19 := FALSE;
   Zulauf_RA_HZS.Bef.Res_20 := FALSE;
   Zulauf_RA_HZS.Bef.Res_21 := FALSE;
   Zulauf_RA_HZS.Bef.Res_22 := FALSE;
   Zulauf_RA_HZS.Bef.Res_23 := FALSE;
   Zulauf_RA_HZS.Bef.Res_24 := FALSE;
   Zulauf_RA_HZS.Bef.Res_25 := FALSE;
   Zulauf_RA_HZS.Bef.Res_26 := FALSE;
   Zulauf_RA_HZS.Bef.Res_27 := FALSE;
   Zulauf_RA_HZS.Bef.Res_28 := FALSE;
   Zulauf_RA_HZS.Bef.Res_29 := FALSE;
   Zulauf_RA_HZS.Bef.BF_Set_SW_chg := FALSE;
   Zulauf_RA_HZS.Bef.BF_Quit := FALSE;
   Zulauf_RA_HZS.SW_Hand := 0.0;
   Zulauf_RA_VKS.Bef.Bed_Res := FALSE;
   Zulauf_RA_VKS.Bef.Bed_UV := FALSE;
   Zulauf_RA_VKS.Bef.Bed_NHV := FALSE;
   Zulauf_RA_VKS.Bef.Bed_PLS := FALSE;
   Zulauf_RA_VKS.Bef.BA_Hand := FALSE;
   Zulauf_RA_VKS.Bef.BA_Auto := FALSE;
   Zulauf_RA_VKS.Bef.BF_Ein1 := FALSE;
   Zulauf_RA_VKS.Bef.BF_Ein2 := FALSE;
   Zulauf_RA_VKS.Bef.BF_Aus := FALSE;
   Zulauf_RA_VKS.Bef.BZ_Res := FALSE;
   Zulauf_RA_VKS.Bef.Res_10 := FALSE;
   Zulauf_RA_VKS.Bef.Res_11 := FALSE;
   Zulauf_RA_VKS.Bef.Res_12 := FALSE;
   Zulauf_RA_VKS.Bef.Res_13 := FALSE;
   Zulauf_RA_VKS.Bef.Res_14 := FALSE;
   Zulauf_RA_VKS.Bef.Res_15 := FALSE;
   Zulauf_RA_VKS.Bef.Res_16 := FALSE;
   Zulauf_RA_VKS.Bef.Res_17 := FALSE;
   Zulauf_RA_VKS.Bef.Res_18 := FALSE;
   Zulauf_RA_VKS.Bef.Res_19 := FALSE;
   Zulauf_RA_VKS.Bef.Res_20 := FALSE;
   Zulauf_RA_VKS.Bef.Res_21 := FALSE;
   Zulauf_RA_VKS.Bef.Res_22 := FALSE;
   Zulauf_RA_VKS.Bef.Res_23 := FALSE;
   Zulauf_RA_VKS.Bef.Res_24 := FALSE;
   Zulauf_RA_VKS.Bef.Res_25 := FALSE;
   Zulauf_RA_VKS.Bef.Res_26 := FALSE;
   Zulauf_RA_VKS.Bef.Res_27 := FALSE;
   Zulauf_RA_VKS.Bef.Res_28 := FALSE;
   Zulauf_RA_VKS.Bef.Res_29 := FALSE;
   Zulauf_RA_VKS.Bef.BF_Set_SW_chg := FALSE;
   Zulauf_RA_VKS.Bef.BF_Quit := FALSE;
   Zulauf_RA_VKS.SW_Hand := 0.0;
   Zulauf_RA_V.Bef.Bed_Res := FALSE;
   Zulauf_RA_V.Bef.Bed_UV := FALSE;
   Zulauf_RA_V.Bef.Bed_NHV := FALSE;
   Zulauf_RA_V.Bef.Bed_PLS := FALSE;
   Zulauf_RA_V.Bef.BA_Hand := FALSE;
   Zulauf_RA_V.Bef.BA_Auto := FALSE;
   Zulauf_RA_V.Bef.BF_Ein1 := FALSE;
   Zulauf_RA_V.Bef.BF_Ein2 := FALSE;
   Zulauf_RA_V.Bef.BF_Aus := FALSE;
   Zulauf_RA_V.Bef.BZ_Res := FALSE;
   Zulauf_RA_V.Bef.Res_10 := FALSE;
   Zulauf_RA_V.Bef.Res_11 := FALSE;
   Zulauf_RA_V.Bef.Res_12 := FALSE;
   Zulauf_RA_V.Bef.Res_13 := FALSE;
   Zulauf_RA_V.Bef.Res_14 := FALSE;
   Zulauf_RA_V.Bef.Res_15 := FALSE;
   Zulauf_RA_V.Bef.Res_16 := FALSE;
   Zulauf_RA_V.Bef.Res_17 := FALSE;
   Zulauf_RA_V.Bef.Res_18 := FALSE;
   Zulauf_RA_V.Bef.Res_19 := FALSE;
   Zulauf_RA_V.Bef.Res_20 := FALSE;
   Zulauf_RA_V.Bef.Res_21 := FALSE;
   Zulauf_RA_V.Bef.Res_22 := FALSE;
   Zulauf_RA_V.Bef.Res_23 := FALSE;
   Zulauf_RA_V.Bef.Res_24 := FALSE;
   Zulauf_RA_V.Bef.Res_25 := FALSE;
   Zulauf_RA_V.Bef.Res_26 := FALSE;
   Zulauf_RA_V.Bef.Res_27 := FALSE;
   Zulauf_RA_V.Bef.Res_28 := FALSE;
   Zulauf_RA_V.Bef.Res_29 := FALSE;
   Zulauf_RA_V.Bef.BF_Set_SW_chg := FALSE;
   Zulauf_RA_V.Bef.BF_Quit := FALSE;
   Zulauf_RA_V.SW_Hand := 0.0;
   Zulauf_RA_RP.Bef.Bed_Res := FALSE;
   Zulauf_RA_RP.Bef.Bed_UV := FALSE;
   Zulauf_RA_RP.Bef.Bed_NHV := FALSE;
   Zulauf_RA_RP.Bef.Bed_PLS := FALSE;
   Zulauf_RA_RP.Bef.BA_Hand := FALSE;
   Zulauf_RA_RP.Bef.BA_Auto := FALSE;
   Zulauf_RA_RP.Bef.BF_Ein1 := FALSE;
   Zulauf_RA_RP.Bef.BF_Ein2 := FALSE;
   Zulauf_RA_RP.Bef.BF_Aus := FALSE;
   Zulauf_RA_RP.Bef.BZ_Res := FALSE;
   Zulauf_RA_RP.Bef.Res_10 := FALSE;
   Zulauf_RA_RP.Bef.Res_11 := FALSE;
   Zulauf_RA_RP.Bef.Res_12 := FALSE;
   Zulauf_RA_RP.Bef.Res_13 := FALSE;
   Zulauf_RA_RP.Bef.Res_14 := FALSE;
   Zulauf_RA_RP.Bef.Res_15 := FALSE;
   Zulauf_RA_RP.Bef.Res_16 := FALSE;
   Zulauf_RA_RP.Bef.Res_17 := FALSE;
   Zulauf_RA_RP.Bef.Res_18 := FALSE;
   Zulauf_RA_RP.Bef.Res_19 := FALSE;
   Zulauf_RA_RP.Bef.Res_20 := FALSE;
   Zulauf_RA_RP.Bef.Res_21 := FALSE;
   Zulauf_RA_RP.Bef.Res_22 := FALSE;
   Zulauf_RA_RP.Bef.Res_23 := FALSE;
   Zulauf_RA_RP.Bef.Res_24 := FALSE;
   Zulauf_RA_RP.Bef.Res_25 := FALSE;
   Zulauf_RA_RP.Bef.Res_26 := FALSE;
   Zulauf_RA_RP.Bef.Res_27 := FALSE;
   Zulauf_RA_RP.Bef.Res_28 := FALSE;
   Zulauf_RA_RP.Bef.Res_29 := FALSE;
   Zulauf_RA_RP.Bef.BF_Set_SW_chg := FALSE;
   Zulauf_RA_RP.Bef.BF_Quit := FALSE;
   Zulauf_RA_RP.SW_Hand := 0.0;
   Zulauf_RA_FP.Bef.Bed_Res := FALSE;
   Zulauf_RA_FP.Bef.Bed_UV := FALSE;
   Zulauf_RA_FP.Bef.Bed_NHV := FALSE;
   Zulauf_RA_FP.Bef.Bed_PLS := FALSE;
   Zulauf_RA_FP.Bef.BA_Hand := FALSE;
   Zulauf_RA_FP.Bef.BA_Auto := FALSE;
   Zulauf_RA_FP.Bef.BF_Ein1 := FALSE;
   Zulauf_RA_FP.Bef.BF_Ein2 := FALSE;
   Zulauf_RA_FP.Bef.BF_Aus := FALSE;
   Zulauf_RA_FP.Bef.BZ_Res := FALSE;
   Zulauf_RA_FP.Bef.Res_10 := FALSE;
   Zulauf_RA_FP.Bef.Res_11 := FALSE;
   Zulauf_RA_FP.Bef.Res_12 := FALSE;
   Zulauf_RA_FP.Bef.Res_13 := FALSE;
   Zulauf_RA_FP.Bef.Res_14 := FALSE;
   Zulauf_RA_FP.Bef.Res_15 := FALSE;
   Zulauf_RA_FP.Bef.Res_16 := FALSE;
   Zulauf_RA_FP.Bef.Res_17 := FALSE;
   Zulauf_RA_FP.Bef.Res_18 := FALSE;
   Zulauf_RA_FP.Bef.Res_19 := FALSE;
   Zulauf_RA_FP.Bef.Res_20 := FALSE;
   Zulauf_RA_FP.Bef.Res_21 := FALSE;
   Zulauf_RA_FP.Bef.Res_22 := FALSE;
   Zulauf_RA_FP.Bef.Res_23 := FALSE;
   Zulauf_RA_FP.Bef.Res_24 := FALSE;
   Zulauf_RA_FP.Bef.Res_25 := FALSE;
   Zulauf_RA_FP.Bef.Res_26 := FALSE;
   Zulauf_RA_FP.Bef.Res_27 := FALSE;
   Zulauf_RA_FP.Bef.Res_28 := FALSE;
   Zulauf_RA_FP.Bef.Res_29 := FALSE;
   Zulauf_RA_FP.Bef.BF_Set_SW_chg := FALSE;
   Zulauf_RA_FP.Bef.BF_Quit := FALSE;
   Zulauf_RA_FP.SW_Hand := 0.0;
   Schlamm_BP.Bef.Bed_Res := FALSE;
   Schlamm_BP.Bef.Bed_UV := FALSE;
   Schlamm_BP.Bef.Bed_NHV := FALSE;
   Schlamm_BP.Bef.Bed_PLS := FALSE;
   Schlamm_BP.Bef.BA_Hand := FALSE;
   Schlamm_BP.Bef.BA_Auto := FALSE;
   Schlamm_BP.Bef.BF_Ein1 := FALSE;
   Schlamm_BP.Bef.BF_Ein2 := FALSE;
   Schlamm_BP.Bef.BF_Aus := FALSE;
   Schlamm_BP.Bef.BZ_Res := FALSE;
   Schlamm_BP.Bef.Res_10 := FALSE;
   Schlamm_BP.Bef.Res_11 := FALSE;
   Schlamm_BP.Bef.Res_12 := FALSE;
   Schlamm_BP.Bef.Res_13 := FALSE;
   Schlamm_BP.Bef.Res_14 := FALSE;
   Schlamm_BP.Bef.Res_15 := FALSE;
   Schlamm_BP.Bef.Res_16 := FALSE;
   Schlamm_BP.Bef.Res_17 := FALSE;
   Schlamm_BP.Bef.Res_18 := FALSE;
   Schlamm_BP.Bef.Res_19 := FALSE;
   Schlamm_BP.Bef.Res_20 := FALSE;
   Schlamm_BP.Bef.Res_21 := FALSE;
   Schlamm_BP.Bef.Res_22 := FALSE;
   Schlamm_BP.Bef.Res_23 := FALSE;
   Schlamm_BP.Bef.Res_24 := FALSE;
   Schlamm_BP.Bef.Res_25 := FALSE;
   Schlamm_BP.Bef.Res_26 := FALSE;
   Schlamm_BP.Bef.Res_27 := FALSE;
   Schlamm_BP.Bef.Res_28 := FALSE;
   Schlamm_BP.Bef.Res_29 := FALSE;
   Schlamm_BP.Bef.BF_Set_SW_chg := FALSE;
   Schlamm_BP.Bef.BF_Quit := FALSE;
   Schlamm_BP.SW_Hand := 0.0;
   Truebwasser_P1.Bef.Bed_Res := FALSE;
   Truebwasser_P1.Bef.Bed_UV := FALSE;
   Truebwasser_P1.Bef.Bed_NHV := FALSE;
   Truebwasser_P1.Bef.Bed_PLS := FALSE;
   Truebwasser_P1.Bef.BA_Hand := FALSE;
   Truebwasser_P1.Bef.BA_Auto := FALSE;
   Truebwasser_P1.Bef.BF_Ein1 := FALSE;
   Truebwasser_P1.Bef.BF_Ein2 := FALSE;
   Truebwasser_P1.Bef.BF_Aus := FALSE;
   Truebwasser_P1.Bef.BZ_Res := FALSE;
   Truebwasser_P1.Bef.Res_10 := FALSE;
   Truebwasser_P1.Bef.Res_11 := FALSE;
   Truebwasser_P1.Bef.Res_12 := FALSE;
   Truebwasser_P1.Bef.Res_13 := FALSE;
   Truebwasser_P1.Bef.Res_14 := FALSE;
   Truebwasser_P1.Bef.Res_15 := FALSE;
   Truebwasser_P1.Bef.Res_16 := FALSE;
   Truebwasser_P1.Bef.Res_17 := FALSE;
   Truebwasser_P1.Bef.Res_18 := FALSE;
   Truebwasser_P1.Bef.Res_19 := FALSE;
   Truebwasser_P1.Bef.Res_20 := FALSE;
   Truebwasser_P1.Bef.Res_21 := FALSE;
   Truebwasser_P1.Bef.Res_22 := FALSE;
   Truebwasser_P1.Bef.Res_23 := FALSE;
   Truebwasser_P1.Bef.Res_24 := FALSE;
   Truebwasser_P1.Bef.Res_25 := FALSE;
   Truebwasser_P1.Bef.Res_26 := FALSE;
   Truebwasser_P1.Bef.Res_27 := FALSE;
   Truebwasser_P1.Bef.Res_28 := FALSE;
   Truebwasser_P1.Bef.Res_29 := FALSE;
   Truebwasser_P1.Bef.BF_Set_SW_chg := FALSE;
   Truebwasser_P1.Bef.BF_Quit := FALSE;
   Truebwasser_P1.SW_Hand := 0.0;
   Truebwasser_P2.Bef.Bed_Res := FALSE;
   Truebwasser_P2.Bef.Bed_UV := FALSE;
   Truebwasser_P2.Bef.Bed_NHV := FALSE;
   Truebwasser_P2.Bef.Bed_PLS := FALSE;
   Truebwasser_P2.Bef.BA_Hand := FALSE;
   Truebwasser_P2.Bef.BA_Auto := FALSE;
   Truebwasser_P2.Bef.BF_Ein1 := FALSE;
   Truebwasser_P2.Bef.BF_Ein2 := FALSE;
   Truebwasser_P2.Bef.BF_Aus := FALSE;
   Truebwasser_P2.Bef.BZ_Res := FALSE;
   Truebwasser_P2.Bef.Res_10 := FALSE;
   Truebwasser_P2.Bef.Res_11 := FALSE;
   Truebwasser_P2.Bef.Res_12 := FALSE;
   Truebwasser_P2.Bef.Res_13 := FALSE;
   Truebwasser_P2.Bef.Res_14 := FALSE;
   Truebwasser_P2.Bef.Res_15 := FALSE;
   Truebwasser_P2.Bef.Res_16 := FALSE;
   Truebwasser_P2.Bef.Res_17 := FALSE;
   Truebwasser_P2.Bef.Res_18 := FALSE;
   Truebwasser_P2.Bef.Res_19 := FALSE;
   Truebwasser_P2.Bef.Res_20 := FALSE;
   Truebwasser_P2.Bef.Res_21 := FALSE;
   Truebwasser_P2.Bef.Res_22 := FALSE;
   Truebwasser_P2.Bef.Res_23 := FALSE;
   Truebwasser_P2.Bef.Res_24 := FALSE;
   Truebwasser_P2.Bef.Res_25 := FALSE;
   Truebwasser_P2.Bef.Res_26 := FALSE;
   Truebwasser_P2.Bef.Res_27 := FALSE;
   Truebwasser_P2.Bef.Res_28 := FALSE;
   Truebwasser_P2.Bef.Res_29 := FALSE;
   Truebwasser_P2.Bef.BF_Set_SW_chg := FALSE;
   Truebwasser_P2.Bef.BF_Quit := FALSE;
   Truebwasser_P2.SW_Hand := 0.0;
   Schlamm_AS.Bef.Bed_Res := FALSE;
   Schlamm_AS.Bef.Bed_UV := FALSE;
   Schlamm_AS.Bef.Bed_NHV := FALSE;
   Schlamm_AS.Bef.Bed_PLS := FALSE;
   Schlamm_AS.Bef.BA_Hand := FALSE;
   Schlamm_AS.Bef.BA_Auto := FALSE;
   Schlamm_AS.Bef.BF_Ein1 := FALSE;
   Schlamm_AS.Bef.BF_Ein2 := FALSE;
   Schlamm_AS.Bef.BF_Aus := FALSE;
   Schlamm_AS.Bef.BZ_Res := FALSE;
   Schlamm_AS.Bef.Res_10 := FALSE;
   Schlamm_AS.Bef.Res_11 := FALSE;
   Schlamm_AS.Bef.Res_12 := FALSE;
   Schlamm_AS.Bef.Res_13 := FALSE;
   Schlamm_AS.Bef.Res_14 := FALSE;
   Schlamm_AS.Bef.Res_15 := FALSE;
   Schlamm_AS.Bef.Res_16 := FALSE;
   Schlamm_AS.Bef.Res_17 := FALSE;
   Schlamm_AS.Bef.Res_18 := FALSE;
   Schlamm_AS.Bef.Res_19 := FALSE;
   Schlamm_AS.Bef.Res_20 := FALSE;
   Schlamm_AS.Bef.Res_21 := FALSE;
   Schlamm_AS.Bef.Res_22 := FALSE;
   Schlamm_AS.Bef.Res_23 := FALSE;
   Schlamm_AS.Bef.Res_24 := FALSE;
   Schlamm_AS.Bef.Res_25 := FALSE;
   Schlamm_AS.Bef.Res_26 := FALSE;
   Schlamm_AS.Bef.Res_27 := FALSE;
   Schlamm_AS.Bef.Res_28 := FALSE;
   Schlamm_AS.Bef.Res_29 := FALSE;
   Schlamm_AS.Bef.BF_Set_SW_chg := FALSE;
   Schlamm_AS.Bef.BF_Quit := FALSE;
   Schlamm_AS.SW_Hand := 0.0;
   BB2_SR_K.Bef.Bed_Res := FALSE;
   BB2_SR_K.Bef.Bed_UV := FALSE;
   BB2_SR_K.Bef.Bed_NHV := FALSE;
   BB2_SR_K.Bef.Bed_PLS := FALSE;
   BB2_SR_K.Bef.BA_Hand := FALSE;
   BB2_SR_K.Bef.BA_Auto := FALSE;
   BB2_SR_K.Bef.BF_Ein1 := FALSE;
   BB2_SR_K.Bef.BF_Ein2 := FALSE;
   BB2_SR_K.Bef.BF_Aus := FALSE;
   BB2_SR_K.Bef.BZ_Res := FALSE;
   BB2_SR_K.Bef.Res_10 := FALSE;
   BB2_SR_K.Bef.Res_11 := FALSE;
   BB2_SR_K.Bef.Res_12 := FALSE;
   BB2_SR_K.Bef.Res_13 := FALSE;
   BB2_SR_K.Bef.Res_14 := FALSE;
   BB2_SR_K.Bef.Res_15 := FALSE;
   BB2_SR_K.Bef.Res_16 := FALSE;
   BB2_SR_K.Bef.Res_17 := FALSE;
   BB2_SR_K.Bef.Res_18 := FALSE;
   BB2_SR_K.Bef.Res_19 := FALSE;
   BB2_SR_K.Bef.Res_20 := FALSE;
   BB2_SR_K.Bef.Res_21 := FALSE;
   BB2_SR_K.Bef.Res_22 := FALSE;
   BB2_SR_K.Bef.Res_23 := FALSE;
   BB2_SR_K.Bef.Res_24 := FALSE;
   BB2_SR_K.Bef.Res_25 := FALSE;
   BB2_SR_K.Bef.Res_26 := FALSE;
   BB2_SR_K.Bef.Res_27 := FALSE;
   BB2_SR_K.Bef.Res_28 := FALSE;
   BB2_SR_K.Bef.Res_29 := FALSE;
   BB2_SR_K.Bef.BF_Set_SW_chg := FALSE;
   BB2_SR_K.Bef.BF_Quit := FALSE;
   BB2_SR_K.SW_Hand := 0.0;

END_DATA_BLOCK

DATA_BLOCK "DB107_Antriebe_EA"
{ S7_Optimized_Access := 'FALSE' }
VERSION : 0.1
NON_RETAIN
   STRUCT
      BB_G1 : "T_ANTRIEB_EA";   // Belebung - Gebläse 1
      BB_G2 : "T_ANTRIEB_EA";   // Belebung - Gebläse 2
      BB_G3 : "T_ANTRIEB_EA";   // Belebung - Gebläse 3
      BB_SHL_G1 : "T_ANTRIEB_EA";   // Belebung - Schallhaubenlüfter Gebläse 1
      BB_SHL_G2 : "T_ANTRIEB_EA";   // Belebung - Schallhaubenlüfter Gebläse 2
      BB_SHL_G3 : "T_ANTRIEB_EA";   // Belebung - Schallhaubenlüfter Gebläse 3
      BB_AV : "T_ANTRIEB_EA";   // Belebung - Gebläsestation - Abluftventilator
      BB_LS1 : "T_ANTRIEB_EA";   // Belebung - Gebläsestation - Luftwegschieber 1
      BB_LS2 : "T_ANTRIEB_EA";   // Belebung - Gebläsestation - Luftwegschieber 2
      BB1_RZP1 : "T_ANTRIEB_EA";   // Becken 1 - Rezipumpe 1
      BB1_RZP2 : "T_ANTRIEB_EA";   // Becken 1 - Rezipumpe 2
      BB1_UeSP : "T_ANTRIEB_EA";   // Becken 1 - ÜSS-Pumpe
      BB1_AS1 : "T_ANTRIEB_EA";   // Becken 1 - Ablaufschieber 1
      BB1_AS2 : "T_ANTRIEB_EA";   // Becken 1 - Ablaufschieber 2
      BB1_SR1 : "T_ANTRIEB_EA";   // Becken 1 - MV Schlammrückführung 1
      BB1_SR2 : "T_ANTRIEB_EA";   // Becken 1 - MV Schlammrückführung 2
      BB2_RZP1 : "T_ANTRIEB_EA";   // Becken 2 - Rezipumpe 1
      BB2_RZP2 : "T_ANTRIEB_EA";   // Becken 2 - Rezipumpe 2
      BB2_UeSP : "T_ANTRIEB_EA";   // Becken 2 - ÜSS-Pumpe
      BB2_AS1 : "T_ANTRIEB_EA";   // Becken 2 - Ablaufschieber 1
      BB2_AS2 : "T_ANTRIEB_EA";   // Becken 2 - Ablaufschieber 2
      BB2_SR1 : "T_ANTRIEB_EA";   // Becken 2 - MV Schlammrückführung 1
      BB2_SR2 : "T_ANTRIEB_EA";   // Becken 2 - MV Schlammrückführung 2
      BB1_SR_K : "T_ANTRIEB_EA";   // Becken 1- Druckluftkompressor Schlammrückführung
      Zulauf_AR_P1 : "T_ANTRIEB_EA";   // Zulauf - Pumpwerk "Alter Rechen" - Pumpe 1
      Zulauf_AR_P2 : "T_ANTRIEB_EA";   // Zulauf - Pumpwerk "Alter Rechen" - Pumpe 2
      Zulauf_AS : "T_ANTRIEB_EA";   // Zulauf - Vorlagebehälter - Absperrschieber
      Zulauf_RA_SA : "T_ANTRIEB_EA";   // Zulauf - Rechen - Sieb
      Zulauf_RA_HZS : "T_ANTRIEB_EA";   // Zulauf - Rechen - HZS
      Zulauf_RA_VKS : "T_ANTRIEB_EA";   // Zulauf - Rechen - VZS
      Zulauf_RA_V : "T_ANTRIEB_EA";   // Zulauf - Rechen - Belüfter
      Zulauf_RA_RP : "T_ANTRIEB_EA";   // Zulauf - Rechen - Räumpaddel
      Zulauf_RA_FP : "T_ANTRIEB_EA";   // Zulauf - Rechen - Fettpumpe
      Schlamm_BP : "T_ANTRIEB_EA";   // Schlamm - Beschickungspumpe Schlammbeete
      Truebwasser_P1 : "T_ANTRIEB_EA";   // Trübwasserpumpwerk - Pumpe 1
      Truebwasser_P2 : "T_ANTRIEB_EA";   // Trübwasserpumpwerk - Pumpe 2
      Schlamm_AS : "T_ANTRIEB_EA";   // Schlamm - Absperrschieber Schlammbeete
      BB2_SR_K : "T_ANTRIEB_EA";   // Becken 2 - Druckluftkompressor Schlammrückführung
      Zulauf_DosP : "T_ANTRIEB_EA";   // Zulauf - Dosierpumpe
   END_STRUCT;


